REGION Network 138: GROUP 6 SAFE STOP 1 DEACTIVATE
   RUNG wire#powerrail
      Contact( "DB1018_SAFETY_TAGS".ALWAYS_ON )
      Coil( "DB1018_SAFETY_TAGS".GROUP_6_E20.SS1_Deactivate )
   END_RUNG
   // the same network as SCL:
   "DB1018_SAFETY_TAGS".GROUP_6_E20.SS1_Deactivate := "DB1018_SAFETY_TAGS".ALWAYS_ON;
END_REGION

REGION Network 139: DESELECT SAFE STOP 1
   RUNG wire#powerrail
      Contact( "DB1018_SAFETY_TAGS".GROUP_6_E20.SS1_Deactivate )
      Coil( "E20_SAFETY_OUT".Deselect_SS1 )
   END_RUNG
   // the same network as SCL:
   "E20_SAFETY_OUT".Deselect_SS1 := "DB1018_SAFETY_TAGS".GROUP_6_E20.SS1_Deactivate;
END_REGION

REGION Network 140: GROUP 6 SAFE STOP 2 DEACTIVATE
   RUNG wire#powerrail
      Contact( "DB1018_SAFETY_TAGS".E_STOP_OK )
      wire#w1
      Coil( "DB1018_SAFETY_TAGS".GROUP_6_E20.SS2_Deactivate )
   END_RUNG
   RUNG wire#powerrail
      Contact( "DB1018_SAFETY_TAGS".SAFE_DOORS_U02_CLOSED_AND_LOCKED )
   END_RUNG wire#w1
   // the same network as SCL:
   "DB1018_SAFETY_TAGS".GROUP_6_E20.SS2_Deactivate := "DB1018_SAFETY_TAGS".E_STOP_OK OR "DB1018_SAFETY_TAGS".SAFE_DOORS_U02_CLOSED_AND_LOCKED;
END_REGION

REGION Network 141: DESELECT SAFE STOP 2
   RUNG wire#powerrail
      Contact( "DB1018_SAFETY_TAGS".GROUP_6_E20.SS2_Deactivate )
      Coil( "E20_SAFETY_OUT".Deselect_SS2 )
   END_RUNG
   // the same network as SCL:
   "E20_SAFETY_OUT".Deselect_SS2 := "DB1018_SAFETY_TAGS".GROUP_6_E20.SS2_Deactivate;
END_REGION

REGION Network 142: GROUP 6 SAFE STOP 2 EXTENDED DEACTIVATE
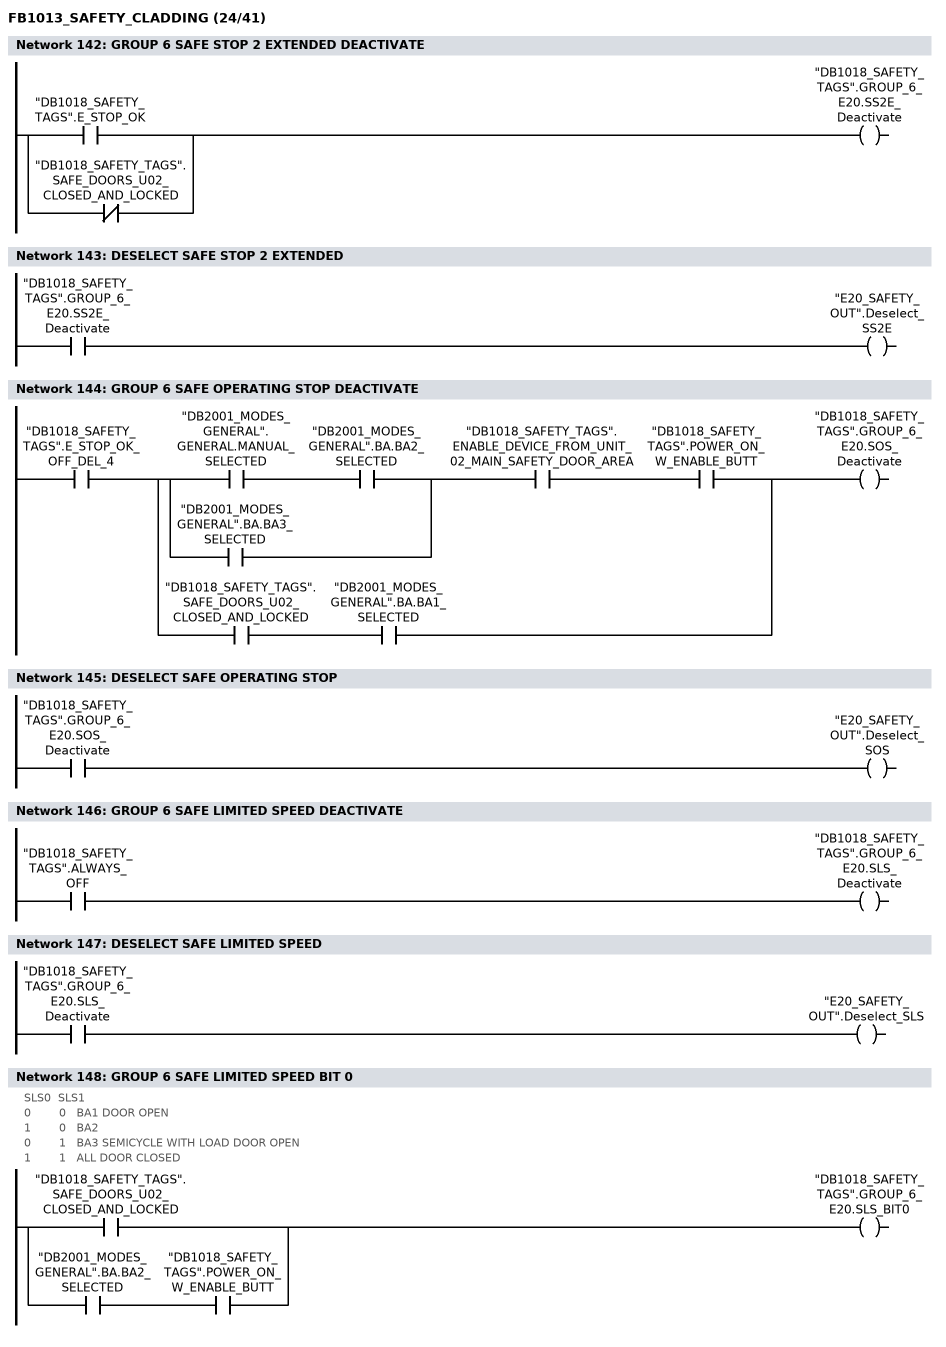
   RUNG wire#powerrail
      Contact( "DB1018_SAFETY_TAGS".E_STOP_OK )
      wire#w1
      Coil( "DB1018_SAFETY_TAGS".GROUP_6_E20.SS2E_Deactivate )
   END_RUNG
   RUNG wire#powerrail
      I_Contact( "DB1018_SAFETY_TAGS".SAFE_DOORS_U02_CLOSED_AND_LOCKED )
   END_RUNG wire#w1
   // the same network as SCL:
   "DB1018_SAFETY_TAGS".GROUP_6_E20.SS2E_Deactivate := "DB1018_SAFETY_TAGS".E_STOP_OK OR NOT "DB1018_SAFETY_TAGS".SAFE_DOORS_U02_CLOSED_AND_LOCKED;
END_REGION

REGION Network 143: DESELECT SAFE STOP 2 EXTENDED
   RUNG wire#powerrail
      Contact( "DB1018_SAFETY_TAGS".GROUP_6_E20.SS2E_Deactivate )
      Coil( "E20_SAFETY_OUT".Deselect_SS2E )
   END_RUNG
   // the same network as SCL:
   "E20_SAFETY_OUT".Deselect_SS2E := "DB1018_SAFETY_TAGS".GROUP_6_E20.SS2E_Deactivate;
END_REGION

REGION Network 144: GROUP 6 SAFE OPERATING STOP DEACTIVATE
   RUNG wire#powerrail
      Contact( "DB1018_SAFETY_TAGS".E_STOP_OK_OFF_DEL_4 )
      wire#w1
      Contact( "DB2001_MODES_GENERAL".GENERAL.MANUAL_SELECTED )
      Contact( "DB2001_MODES_GENERAL".BA.BA2_SELECTED )
      wire#w2
      Contact( "DB1018_SAFETY_TAGS".ENABLE_DEVICE_FROM_UNIT_02_MAIN_SAFETY_DOOR_AREA )
      Contact( "DB1018_SAFETY_TAGS".POWER_ON_W_ENABLE_BUTT )
      wire#w3
      Coil( "DB1018_SAFETY_TAGS".GROUP_6_E20.SOS_Deactivate )
   END_RUNG
   RUNG wire#w1
      Contact( "DB2001_MODES_GENERAL".BA.BA3_SELECTED )
   END_RUNG wire#w2
   RUNG wire#w1
      Contact( "DB1018_SAFETY_TAGS".SAFE_DOORS_U02_CLOSED_AND_LOCKED )
      Contact( "DB2001_MODES_GENERAL".BA.BA1_SELECTED )
   END_RUNG wire#w3
   // the same network as SCL:
   "DB1018_SAFETY_TAGS".GROUP_6_E20.SOS_Deactivate := "DB1018_SAFETY_TAGS".E_STOP_OK_OFF_DEL_4 AND (((("DB2001_MODES_GENERAL".GENERAL.MANUAL_SELECTED AND "DB2001_MODES_GENERAL".BA.BA2_SELECTED) OR "DB2001_MODES_GENERAL".BA.BA3_SELECTED) AND "DB1018_SAFETY_TAGS".ENABLE_DEVICE_FROM_UNIT_02_MAIN_SAFETY_DOOR_AREA AND "DB1018_SAFETY_TAGS".POWER_ON_W_ENABLE_BUTT) OR ("DB1018_SAFETY_TAGS".SAFE_DOORS_U02_CLOSED_AND_LOCKED AND "DB2001_MODES_GENERAL".BA.BA1_SELECTED));
END_REGION

REGION Network 145: DESELECT SAFE OPERATING STOP
   RUNG wire#powerrail
      Contact( "DB1018_SAFETY_TAGS".GROUP_6_E20.SOS_Deactivate )
      Coil( "E20_SAFETY_OUT".Deselect_SOS )
   END_RUNG
   // the same network as SCL:
   "E20_SAFETY_OUT".Deselect_SOS := "DB1018_SAFETY_TAGS".GROUP_6_E20.SOS_Deactivate;
END_REGION

REGION Network 146: GROUP 6 SAFE LIMITED SPEED DEACTIVATE
   RUNG wire#powerrail
      Contact( "DB1018_SAFETY_TAGS".ALWAYS_OFF )
      Coil( "DB1018_SAFETY_TAGS".GROUP_6_E20.SLS_Deactivate )
   END_RUNG
   // the same network as SCL:
   "DB1018_SAFETY_TAGS".GROUP_6_E20.SLS_Deactivate := "DB1018_SAFETY_TAGS".ALWAYS_OFF;
END_REGION

REGION Network 147: DESELECT SAFE LIMITED SPEED
   RUNG wire#powerrail
      Contact( "DB1018_SAFETY_TAGS".GROUP_6_E20.SLS_Deactivate )
      Coil( "E20_SAFETY_OUT".Deselect_SLS )
   END_RUNG
   // the same network as SCL:
   "E20_SAFETY_OUT".Deselect_SLS := "DB1018_SAFETY_TAGS".GROUP_6_E20.SLS_Deactivate;
END_REGION

REGION Network 148: GROUP 6 SAFE LIMITED SPEED BIT 0
   // SLS0  SLS1
   //    0        0   BA1 DOOR OPEN
   //    1        0   BA2
   //    0        1   BA3 SEMICYCLE WITH LOAD DOOR OPEN
   //    1        1   ALL DOOR CLOSED
   RUNG wire#powerrail
      Contact( "DB1018_SAFETY_TAGS".SAFE_DOORS_U02_CLOSED_AND_LOCKED )
      wire#w1
      Coil( "DB1018_SAFETY_TAGS".GROUP_6_E20.SLS_BIT0 )
   END_RUNG
   RUNG wire#powerrail
      Contact( "DB2001_MODES_GENERAL".BA.BA2_SELECTED )
      Contact( "DB1018_SAFETY_TAGS".POWER_ON_W_ENABLE_BUTT )
   END_RUNG wire#w1
   // the same network as SCL:
   "DB1018_SAFETY_TAGS".GROUP_6_E20.SLS_BIT0 := "DB1018_SAFETY_TAGS".SAFE_DOORS_U02_CLOSED_AND_LOCKED OR ("DB2001_MODES_GENERAL".BA.BA2_SELECTED AND "DB1018_SAFETY_TAGS".POWER_ON_W_ENABLE_BUTT);
END_REGION

REGION Network 149: SELECT SAFE LIMITED SPEED BIT 0
   // SLS0  SLS1
   //    0        0   BA1 DOOR OPEN
   //    1        0   BA2
   //    0        1   BA3 SEMICYCLE WITH LOAD DOOR OPEN
   //    1        1   ALL DOOR CLOSED
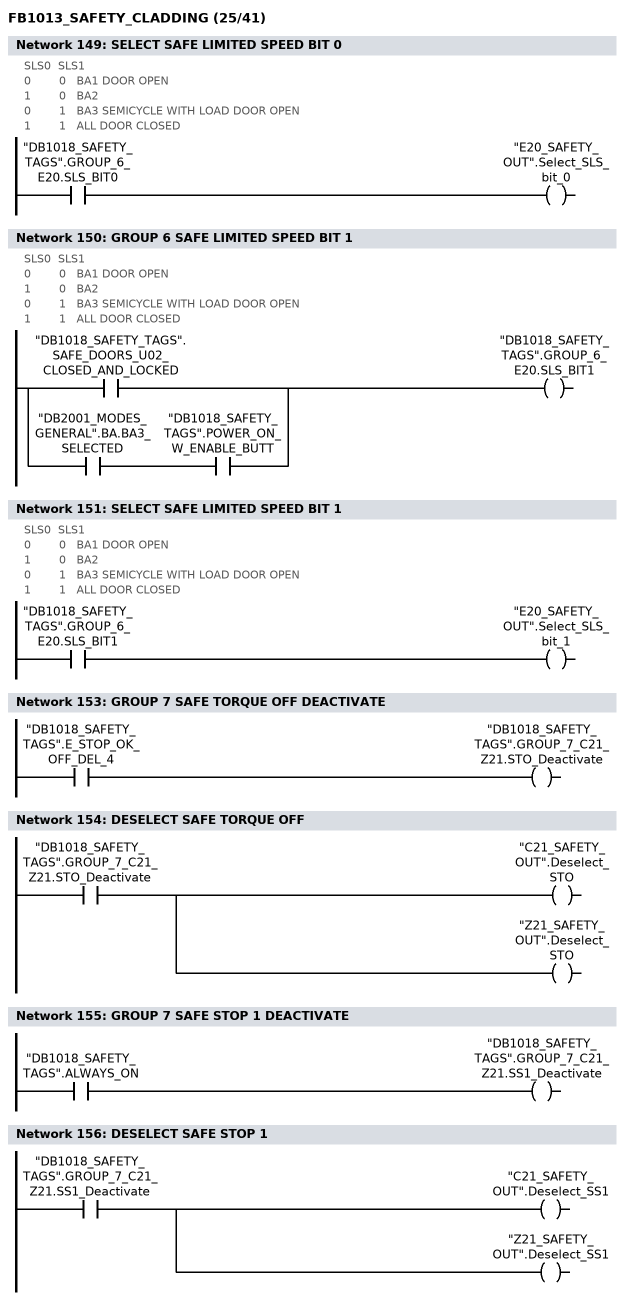
   RUNG wire#powerrail
      Contact( "DB1018_SAFETY_TAGS".GROUP_6_E20.SLS_BIT0 )
      Coil( "E20_SAFETY_OUT".Select_SLS_bit_0 )
   END_RUNG
   // the same network as SCL:
   "E20_SAFETY_OUT".Select_SLS_bit_0 := "DB1018_SAFETY_TAGS".GROUP_6_E20.SLS_BIT0;
END_REGION

REGION Network 150: GROUP 6 SAFE LIMITED SPEED BIT 1
   // SLS0  SLS1
   //    0        0   BA1 DOOR OPEN
   //    1        0   BA2
   //    0        1   BA3 SEMICYCLE WITH LOAD DOOR OPEN
   //    1        1   ALL DOOR CLOSED
   RUNG wire#powerrail
      Contact( "DB1018_SAFETY_TAGS".SAFE_DOORS_U02_CLOSED_AND_LOCKED )
      wire#w1
      Coil( "DB1018_SAFETY_TAGS".GROUP_6_E20.SLS_BIT1 )
   END_RUNG
   RUNG wire#powerrail
      Contact( "DB2001_MODES_GENERAL".BA.BA3_SELECTED )
      Contact( "DB1018_SAFETY_TAGS".POWER_ON_W_ENABLE_BUTT )
   END_RUNG wire#w1
   // the same network as SCL:
   "DB1018_SAFETY_TAGS".GROUP_6_E20.SLS_BIT1 := "DB1018_SAFETY_TAGS".SAFE_DOORS_U02_CLOSED_AND_LOCKED OR ("DB2001_MODES_GENERAL".BA.BA3_SELECTED AND "DB1018_SAFETY_TAGS".POWER_ON_W_ENABLE_BUTT);
END_REGION

REGION Network 151: SELECT SAFE LIMITED SPEED BIT 1
   // SLS0  SLS1
   //    0        0   BA1 DOOR OPEN
   //    1        0   BA2
   //    0        1   BA3 SEMICYCLE WITH LOAD DOOR OPEN
   //    1        1   ALL DOOR CLOSED
   RUNG wire#powerrail
      Contact( "DB1018_SAFETY_TAGS".GROUP_6_E20.SLS_BIT1 )
      Coil( "E20_SAFETY_OUT".Select_SLS_bit_1 )
   END_RUNG
   // the same network as SCL:
   "E20_SAFETY_OUT".Select_SLS_bit_1 := "DB1018_SAFETY_TAGS".GROUP_6_E20.SLS_BIT1;
END_REGION

REGION Network 152: *************** GROUP 7 - C21 / Z21 ***************
END_REGION

REGION Network 153: GROUP 7 SAFE TORQUE OFF DEACTIVATE
   RUNG wire#powerrail
      Contact( "DB1018_SAFETY_TAGS".E_STOP_OK_OFF_DEL_4 )
      Coil( "DB1018_SAFETY_TAGS".GROUP_7_C21_Z21.STO_Deactivate )
   END_RUNG
   // the same network as SCL:
   "DB1018_SAFETY_TAGS".GROUP_7_C21_Z21.STO_Deactivate := "DB1018_SAFETY_TAGS".E_STOP_OK_OFF_DEL_4;
END_REGION

REGION Network 154: DESELECT SAFE TORQUE OFF
   RUNG wire#powerrail
      Contact( "DB1018_SAFETY_TAGS".GROUP_7_C21_Z21.STO_Deactivate )
      wire#w1
      Coil( "C21_SAFETY_OUT".Deselect_STO )
   END_RUNG
   RUNG wire#w1
      Coil( "Z21_SAFETY_OUT".Deselect_STO )
   END_RUNG
   // the same network as SCL:
   "C21_SAFETY_OUT".Deselect_STO := "DB1018_SAFETY_TAGS".GROUP_7_C21_Z21.STO_Deactivate;
   "Z21_SAFETY_OUT".Deselect_STO := "DB1018_SAFETY_TAGS".GROUP_7_C21_Z21.STO_Deactivate;
END_REGION

REGION Network 155: GROUP 7 SAFE STOP 1 DEACTIVATE
   RUNG wire#powerrail
      Contact( "DB1018_SAFETY_TAGS".ALWAYS_ON )
      Coil( "DB1018_SAFETY_TAGS".GROUP_7_C21_Z21.SS1_Deactivate )
   END_RUNG
   // the same network as SCL:
   "DB1018_SAFETY_TAGS".GROUP_7_C21_Z21.SS1_Deactivate := "DB1018_SAFETY_TAGS".ALWAYS_ON;
END_REGION

REGION Network 156: DESELECT SAFE STOP 1
   RUNG wire#powerrail
      Contact( "DB1018_SAFETY_TAGS".GROUP_7_C21_Z21.SS1_Deactivate )
      wire#w1
      Coil( "C21_SAFETY_OUT".Deselect_SS1 )
   END_RUNG
   RUNG wire#w1
      Coil( "Z21_SAFETY_OUT".Deselect_SS1 )
   END_RUNG
   // the same network as SCL:
   "C21_SAFETY_OUT".Deselect_SS1 := "DB1018_SAFETY_TAGS".GROUP_7_C21_Z21.SS1_Deactivate;
   "Z21_SAFETY_OUT".Deselect_SS1 := "DB1018_SAFETY_TAGS".GROUP_7_C21_Z21.SS1_Deactivate;
END_REGION

REGION Network 157: GROUP 7 SAFE STOP 2 DEACTIVATE
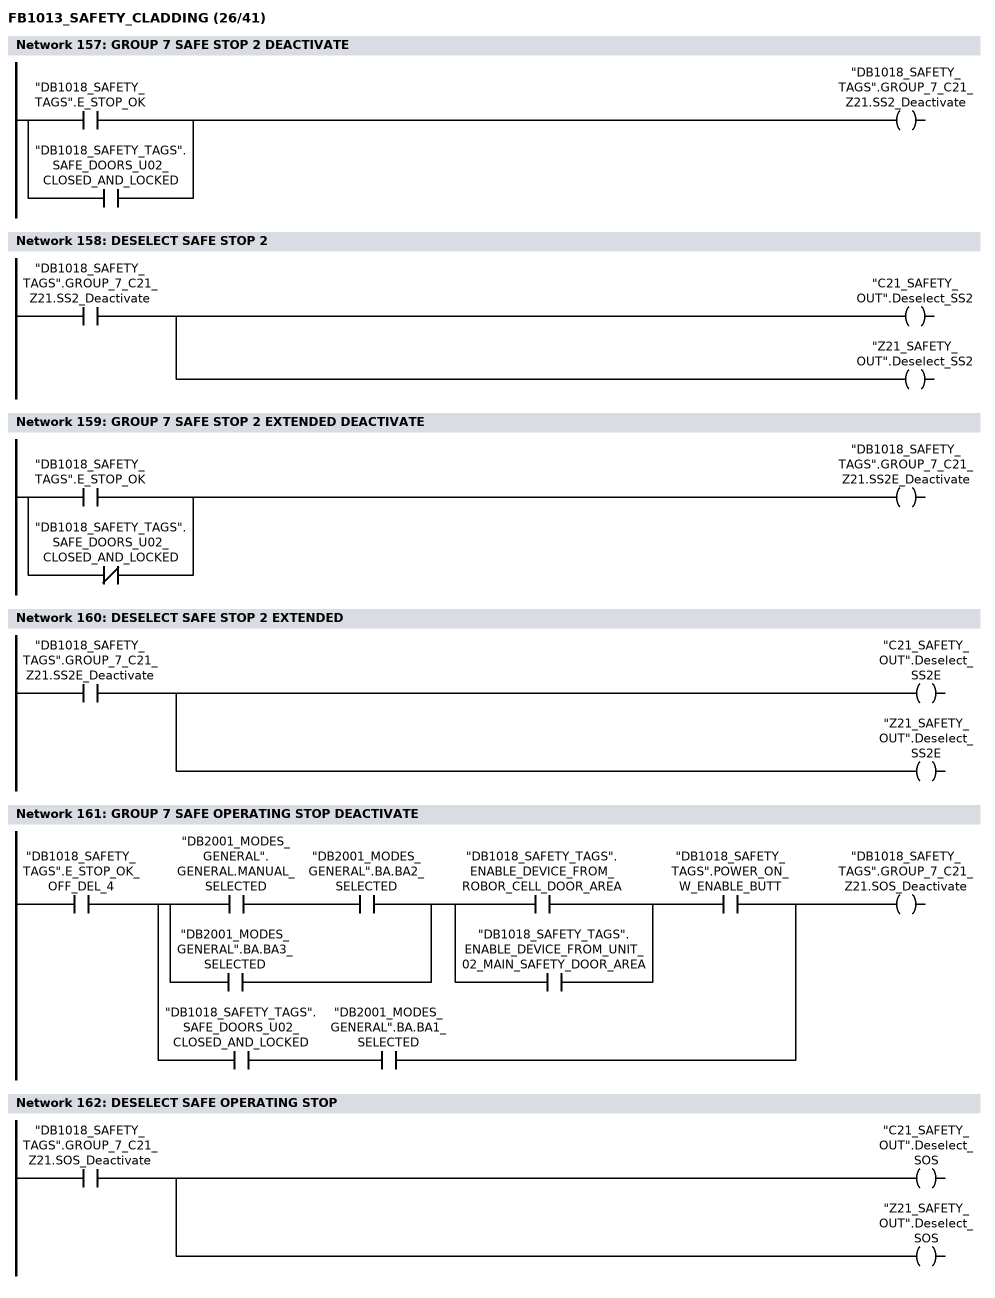
   RUNG wire#powerrail
      Contact( "DB1018_SAFETY_TAGS".E_STOP_OK )
      wire#w1
      Coil( "DB1018_SAFETY_TAGS".GROUP_7_C21_Z21.SS2_Deactivate )
   END_RUNG
   RUNG wire#powerrail
      Contact( "DB1018_SAFETY_TAGS".SAFE_DOORS_U02_CLOSED_AND_LOCKED )
   END_RUNG wire#w1
   // the same network as SCL:
   "DB1018_SAFETY_TAGS".GROUP_7_C21_Z21.SS2_Deactivate := "DB1018_SAFETY_TAGS".E_STOP_OK OR "DB1018_SAFETY_TAGS".SAFE_DOORS_U02_CLOSED_AND_LOCKED;
END_REGION

REGION Network 158: DESELECT SAFE STOP 2
   RUNG wire#powerrail
      Contact( "DB1018_SAFETY_TAGS".GROUP_7_C21_Z21.SS2_Deactivate )
      wire#w1
      Coil( "C21_SAFETY_OUT".Deselect_SS2 )
   END_RUNG
   RUNG wire#w1
      Coil( "Z21_SAFETY_OUT".Deselect_SS2 )
   END_RUNG
   // the same network as SCL:
   "C21_SAFETY_OUT".Deselect_SS2 := "DB1018_SAFETY_TAGS".GROUP_7_C21_Z21.SS2_Deactivate;
   "Z21_SAFETY_OUT".Deselect_SS2 := "DB1018_SAFETY_TAGS".GROUP_7_C21_Z21.SS2_Deactivate;
END_REGION

REGION Network 159: GROUP 7 SAFE STOP 2 EXTENDED DEACTIVATE
   RUNG wire#powerrail
      Contact( "DB1018_SAFETY_TAGS".E_STOP_OK )
      wire#w1
      Coil( "DB1018_SAFETY_TAGS".GROUP_7_C21_Z21.SS2E_Deactivate )
   END_RUNG
   RUNG wire#powerrail
      I_Contact( "DB1018_SAFETY_TAGS".SAFE_DOORS_U02_CLOSED_AND_LOCKED )
   END_RUNG wire#w1
   // the same network as SCL:
   "DB1018_SAFETY_TAGS".GROUP_7_C21_Z21.SS2E_Deactivate := "DB1018_SAFETY_TAGS".E_STOP_OK OR NOT "DB1018_SAFETY_TAGS".SAFE_DOORS_U02_CLOSED_AND_LOCKED;
END_REGION

REGION Network 160: DESELECT SAFE STOP 2 EXTENDED
   RUNG wire#powerrail
      Contact( "DB1018_SAFETY_TAGS".GROUP_7_C21_Z21.SS2E_Deactivate )
      wire#w1
      Coil( "C21_SAFETY_OUT".Deselect_SS2E )
   END_RUNG
   RUNG wire#w1
      Coil( "Z21_SAFETY_OUT".Deselect_SS2E )
   END_RUNG
   // the same network as SCL:
   "C21_SAFETY_OUT".Deselect_SS2E := "DB1018_SAFETY_TAGS".GROUP_7_C21_Z21.SS2E_Deactivate;
   "Z21_SAFETY_OUT".Deselect_SS2E := "DB1018_SAFETY_TAGS".GROUP_7_C21_Z21.SS2E_Deactivate;
END_REGION

REGION Network 161: GROUP 7 SAFE OPERATING STOP DEACTIVATE
   RUNG wire#powerrail
      Contact( "DB1018_SAFETY_TAGS".E_STOP_OK_OFF_DEL_4 )
      wire#w1
      Contact( "DB2001_MODES_GENERAL".GENERAL.MANUAL_SELECTED )
      Contact( "DB2001_MODES_GENERAL".BA.BA2_SELECTED )
      wire#w2
      Contact( "DB1018_SAFETY_TAGS".ENABLE_DEVICE_FROM_ROBOR_CELL_DOOR_AREA )
      wire#w3
      Contact( "DB1018_SAFETY_TAGS".POWER_ON_W_ENABLE_BUTT )
      wire#w4
      Coil( "DB1018_SAFETY_TAGS".GROUP_7_C21_Z21.SOS_Deactivate )
   END_RUNG
   RUNG wire#w1
      Contact( "DB2001_MODES_GENERAL".BA.BA3_SELECTED )
   END_RUNG wire#w2
   RUNG wire#w2
      Contact( "DB1018_SAFETY_TAGS".ENABLE_DEVICE_FROM_UNIT_02_MAIN_SAFETY_DOOR_AREA )
   END_RUNG wire#w3
   RUNG wire#w1
      Contact( "DB1018_SAFETY_TAGS".SAFE_DOORS_U02_CLOSED_AND_LOCKED )
      Contact( "DB2001_MODES_GENERAL".BA.BA1_SELECTED )
   END_RUNG wire#w4
   // the same network as SCL:
   "DB1018_SAFETY_TAGS".GROUP_7_C21_Z21.SOS_Deactivate := "DB1018_SAFETY_TAGS".E_STOP_OK_OFF_DEL_4 AND (((("DB2001_MODES_GENERAL".GENERAL.MANUAL_SELECTED AND "DB2001_MODES_GENERAL".BA.BA2_SELECTED) OR "DB2001_MODES_GENERAL".BA.BA3_SELECTED) AND ("DB1018_SAFETY_TAGS".ENABLE_DEVICE_FROM_ROBOR_CELL_DOOR_AREA OR "DB1018_SAFETY_TAGS".ENABLE_DEVICE_FROM_UNIT_02_MAIN_SAFETY_DOOR_AREA) AND "DB1018_SAFETY_TAGS".POWER_ON_W_ENABLE_BUTT) OR ("DB1018_SAFETY_TAGS".SAFE_DOORS_U02_CLOSED_AND_LOCKED AND "DB2001_MODES_GENERAL".BA.BA1_SELECTED));
END_REGION

REGION Network 162: DESELECT SAFE OPERATING STOP
   RUNG wire#powerrail
      Contact( "DB1018_SAFETY_TAGS".GROUP_7_C21_Z21.SOS_Deactivate )
      wire#w1
      Coil( "C21_SAFETY_OUT".Deselect_SOS )
   END_RUNG
   RUNG wire#w1
      Coil( "Z21_SAFETY_OUT".Deselect_SOS )
   END_RUNG
   // the same network as SCL:
   "C21_SAFETY_OUT".Deselect_SOS := "DB1018_SAFETY_TAGS".GROUP_7_C21_Z21.SOS_Deactivate;
   "Z21_SAFETY_OUT".Deselect_SOS := "DB1018_SAFETY_TAGS".GROUP_7_C21_Z21.SOS_Deactivate;
END_REGION

REGION Network 163: GROUP 7 SAFE LIMITED SPEED DEACTIVATE
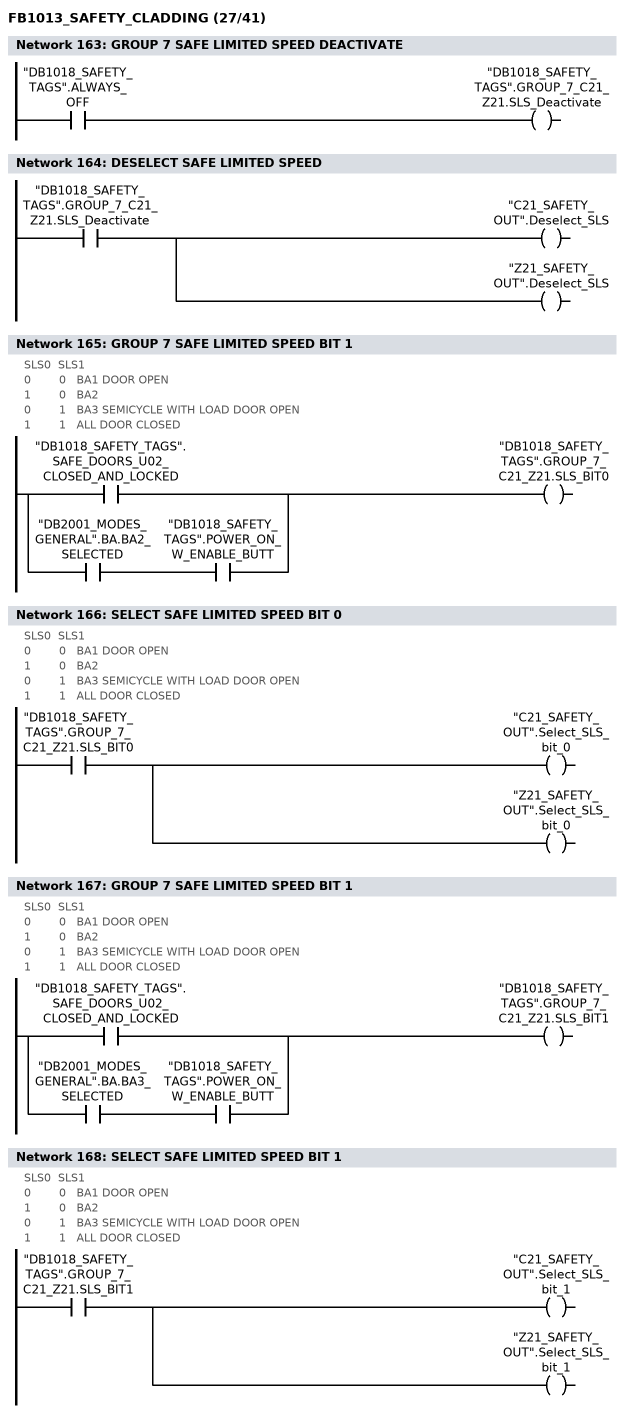
   RUNG wire#powerrail
      Contact( "DB1018_SAFETY_TAGS".ALWAYS_OFF )
      Coil( "DB1018_SAFETY_TAGS".GROUP_7_C21_Z21.SLS_Deactivate )
   END_RUNG
   // the same network as SCL:
   "DB1018_SAFETY_TAGS".GROUP_7_C21_Z21.SLS_Deactivate := "DB1018_SAFETY_TAGS".ALWAYS_OFF;
END_REGION

REGION Network 164: DESELECT SAFE LIMITED SPEED
   RUNG wire#powerrail
      Contact( "DB1018_SAFETY_TAGS".GROUP_7_C21_Z21.SLS_Deactivate )
      wire#w1
      Coil( "C21_SAFETY_OUT".Deselect_SLS )
   END_RUNG
   RUNG wire#w1
      Coil( "Z21_SAFETY_OUT".Deselect_SLS )
   END_RUNG
   // the same network as SCL:
   "C21_SAFETY_OUT".Deselect_SLS := "DB1018_SAFETY_TAGS".GROUP_7_C21_Z21.SLS_Deactivate;
   "Z21_SAFETY_OUT".Deselect_SLS := "DB1018_SAFETY_TAGS".GROUP_7_C21_Z21.SLS_Deactivate;
END_REGION

REGION Network 165: GROUP 7 SAFE LIMITED SPEED BIT 1
   // SLS0  SLS1
   //    0        0   BA1 DOOR OPEN
   //    1        0   BA2
   //    0        1   BA3 SEMICYCLE WITH LOAD DOOR OPEN
   //    1        1   ALL DOOR CLOSED
   RUNG wire#powerrail
      Contact( "DB1018_SAFETY_TAGS".SAFE_DOORS_U02_CLOSED_AND_LOCKED )
      wire#w1
      Coil( "DB1018_SAFETY_TAGS".GROUP_7_C21_Z21.SLS_BIT0 )
   END_RUNG
   RUNG wire#powerrail
      Contact( "DB2001_MODES_GENERAL".BA.BA2_SELECTED )
      Contact( "DB1018_SAFETY_TAGS".POWER_ON_W_ENABLE_BUTT )
   END_RUNG wire#w1
   // the same network as SCL:
   "DB1018_SAFETY_TAGS".GROUP_7_C21_Z21.SLS_BIT0 := "DB1018_SAFETY_TAGS".SAFE_DOORS_U02_CLOSED_AND_LOCKED OR ("DB2001_MODES_GENERAL".BA.BA2_SELECTED AND "DB1018_SAFETY_TAGS".POWER_ON_W_ENABLE_BUTT);
END_REGION

REGION Network 166: SELECT SAFE LIMITED SPEED BIT 0
   // SLS0  SLS1
   //    0        0   BA1 DOOR OPEN
   //    1        0   BA2
   //    0        1   BA3 SEMICYCLE WITH LOAD DOOR OPEN
   //    1        1   ALL DOOR CLOSED
   RUNG wire#powerrail
      Contact( "DB1018_SAFETY_TAGS".GROUP_7_C21_Z21.SLS_BIT0 )
      wire#w1
      Coil( "C21_SAFETY_OUT".Select_SLS_bit_0 )
   END_RUNG
   RUNG wire#w1
      Coil( "Z21_SAFETY_OUT".Select_SLS_bit_0 )
   END_RUNG
   // the same network as SCL:
   "C21_SAFETY_OUT".Select_SLS_bit_0 := "DB1018_SAFETY_TAGS".GROUP_7_C21_Z21.SLS_BIT0;
   "Z21_SAFETY_OUT".Select_SLS_bit_0 := "DB1018_SAFETY_TAGS".GROUP_7_C21_Z21.SLS_BIT0;
END_REGION

REGION Network 167: GROUP 7 SAFE LIMITED SPEED BIT 1
   // SLS0  SLS1
   //    0        0   BA1 DOOR OPEN
   //    1        0   BA2
   //    0        1   BA3 SEMICYCLE WITH LOAD DOOR OPEN
   //    1        1   ALL DOOR CLOSED
   RUNG wire#powerrail
      Contact( "DB1018_SAFETY_TAGS".SAFE_DOORS_U02_CLOSED_AND_LOCKED )
      wire#w1
      Coil( "DB1018_SAFETY_TAGS".GROUP_7_C21_Z21.SLS_BIT1 )
   END_RUNG
   RUNG wire#powerrail
      Contact( "DB2001_MODES_GENERAL".BA.BA3_SELECTED )
      Contact( "DB1018_SAFETY_TAGS".POWER_ON_W_ENABLE_BUTT )
   END_RUNG wire#w1
   // the same network as SCL:
   "DB1018_SAFETY_TAGS".GROUP_7_C21_Z21.SLS_BIT1 := "DB1018_SAFETY_TAGS".SAFE_DOORS_U02_CLOSED_AND_LOCKED OR ("DB2001_MODES_GENERAL".BA.BA3_SELECTED AND "DB1018_SAFETY_TAGS".POWER_ON_W_ENABLE_BUTT);
END_REGION

REGION Network 168: SELECT SAFE LIMITED SPEED BIT 1
   // SLS0  SLS1
   //    0        0   BA1 DOOR OPEN
   //    1        0   BA2
   //    0        1   BA3 SEMICYCLE WITH LOAD DOOR OPEN
   //    1        1   ALL DOOR CLOSED
   RUNG wire#powerrail
      Contact( "DB1018_SAFETY_TAGS".GROUP_7_C21_Z21.SLS_BIT1 )
      wire#w1
      Coil( "C21_SAFETY_OUT".Select_SLS_bit_1 )
   END_RUNG
   RUNG wire#w1
      Coil( "Z21_SAFETY_OUT".Select_SLS_bit_1 )
   END_RUNG
   // the same network as SCL:
   "C21_SAFETY_OUT".Select_SLS_bit_1 := "DB1018_SAFETY_TAGS".GROUP_7_C21_Z21.SLS_BIT1;
   "Z21_SAFETY_OUT".Select_SLS_bit_1 := "DB1018_SAFETY_TAGS".GROUP_7_C21_Z21.SLS_BIT1;
END_REGION

REGION Network 169: *************** GROUP 8 - C22 ***************
END_REGION

REGION Network 170: GROUP 8 SAFE TORQUE OFF DEACTIVATE
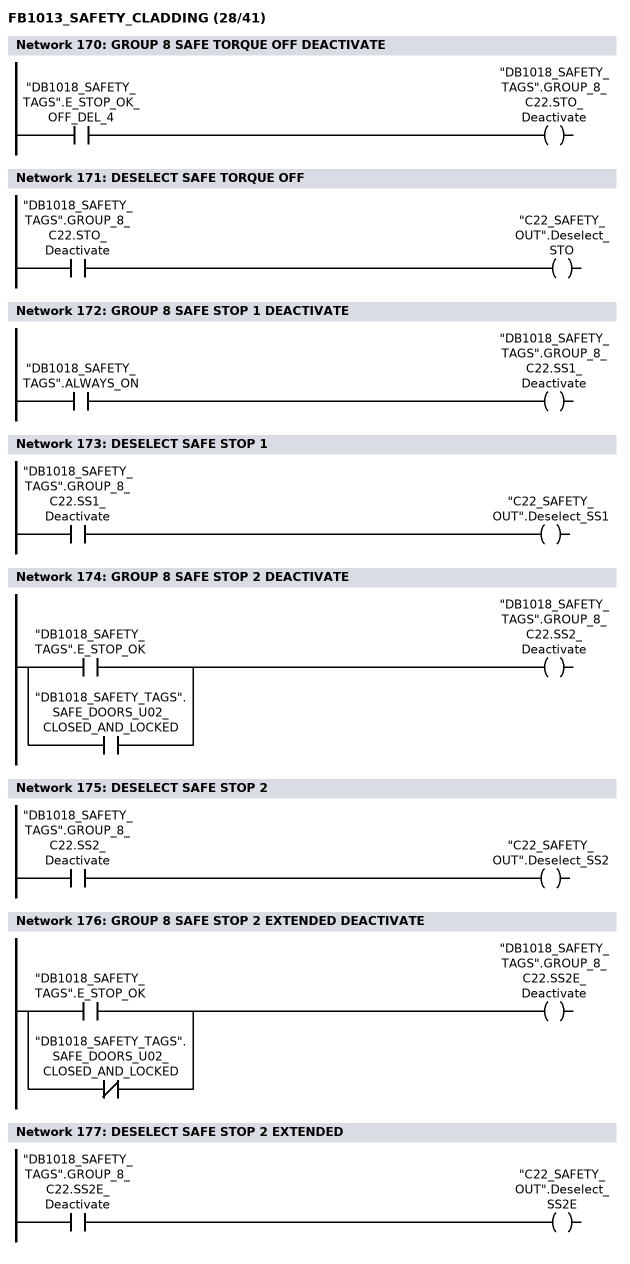
   RUNG wire#powerrail
      Contact( "DB1018_SAFETY_TAGS".E_STOP_OK_OFF_DEL_4 )
      Coil( "DB1018_SAFETY_TAGS".GROUP_8_C22.STO_Deactivate )
   END_RUNG
   // the same network as SCL:
   "DB1018_SAFETY_TAGS".GROUP_8_C22.STO_Deactivate := "DB1018_SAFETY_TAGS".E_STOP_OK_OFF_DEL_4;
END_REGION

REGION Network 171: DESELECT SAFE TORQUE OFF
   RUNG wire#powerrail
      Contact( "DB1018_SAFETY_TAGS".GROUP_8_C22.STO_Deactivate )
      Coil( "C22_SAFETY_OUT".Deselect_STO )
   END_RUNG
   // the same network as SCL:
   "C22_SAFETY_OUT".Deselect_STO := "DB1018_SAFETY_TAGS".GROUP_8_C22.STO_Deactivate;
END_REGION

REGION Network 172: GROUP 8 SAFE STOP 1 DEACTIVATE
   RUNG wire#powerrail
      Contact( "DB1018_SAFETY_TAGS".ALWAYS_ON )
      Coil( "DB1018_SAFETY_TAGS".GROUP_8_C22.SS1_Deactivate )
   END_RUNG
   // the same network as SCL:
   "DB1018_SAFETY_TAGS".GROUP_8_C22.SS1_Deactivate := "DB1018_SAFETY_TAGS".ALWAYS_ON;
END_REGION

REGION Network 173: DESELECT SAFE STOP 1
   RUNG wire#powerrail
      Contact( "DB1018_SAFETY_TAGS".GROUP_8_C22.SS1_Deactivate )
      Coil( "C22_SAFETY_OUT".Deselect_SS1 )
   END_RUNG
   // the same network as SCL:
   "C22_SAFETY_OUT".Deselect_SS1 := "DB1018_SAFETY_TAGS".GROUP_8_C22.SS1_Deactivate;
END_REGION

REGION Network 174: GROUP 8 SAFE STOP 2 DEACTIVATE
   RUNG wire#powerrail
      Contact( "DB1018_SAFETY_TAGS".E_STOP_OK )
      wire#w1
      Coil( "DB1018_SAFETY_TAGS".GROUP_8_C22.SS2_Deactivate )
   END_RUNG
   RUNG wire#powerrail
      Contact( "DB1018_SAFETY_TAGS".SAFE_DOORS_U02_CLOSED_AND_LOCKED )
   END_RUNG wire#w1
   // the same network as SCL:
   "DB1018_SAFETY_TAGS".GROUP_8_C22.SS2_Deactivate := "DB1018_SAFETY_TAGS".E_STOP_OK OR "DB1018_SAFETY_TAGS".SAFE_DOORS_U02_CLOSED_AND_LOCKED;
END_REGION

REGION Network 175: DESELECT SAFE STOP 2
   RUNG wire#powerrail
      Contact( "DB1018_SAFETY_TAGS".GROUP_8_C22.SS2_Deactivate )
      Coil( "C22_SAFETY_OUT".Deselect_SS2 )
   END_RUNG
   // the same network as SCL:
   "C22_SAFETY_OUT".Deselect_SS2 := "DB1018_SAFETY_TAGS".GROUP_8_C22.SS2_Deactivate;
END_REGION

REGION Network 176: GROUP 8 SAFE STOP 2 EXTENDED DEACTIVATE
   RUNG wire#powerrail
      Contact( "DB1018_SAFETY_TAGS".E_STOP_OK )
      wire#w1
      Coil( "DB1018_SAFETY_TAGS".GROUP_8_C22.SS2E_Deactivate )
   END_RUNG
   RUNG wire#powerrail
      I_Contact( "DB1018_SAFETY_TAGS".SAFE_DOORS_U02_CLOSED_AND_LOCKED )
   END_RUNG wire#w1
   // the same network as SCL:
   "DB1018_SAFETY_TAGS".GROUP_8_C22.SS2E_Deactivate := "DB1018_SAFETY_TAGS".E_STOP_OK OR NOT "DB1018_SAFETY_TAGS".SAFE_DOORS_U02_CLOSED_AND_LOCKED;
END_REGION

REGION Network 177: DESELECT SAFE STOP 2 EXTENDED
   RUNG wire#powerrail
      Contact( "DB1018_SAFETY_TAGS".GROUP_8_C22.SS2E_Deactivate )
      Coil( "C22_SAFETY_OUT".Deselect_SS2E )
   END_RUNG
   // the same network as SCL:
   "C22_SAFETY_OUT".Deselect_SS2E := "DB1018_SAFETY_TAGS".GROUP_8_C22.SS2E_Deactivate;
END_REGION

REGION Network 178: GROUP 8 SAFE OPERATING STOP DEACTIVATE
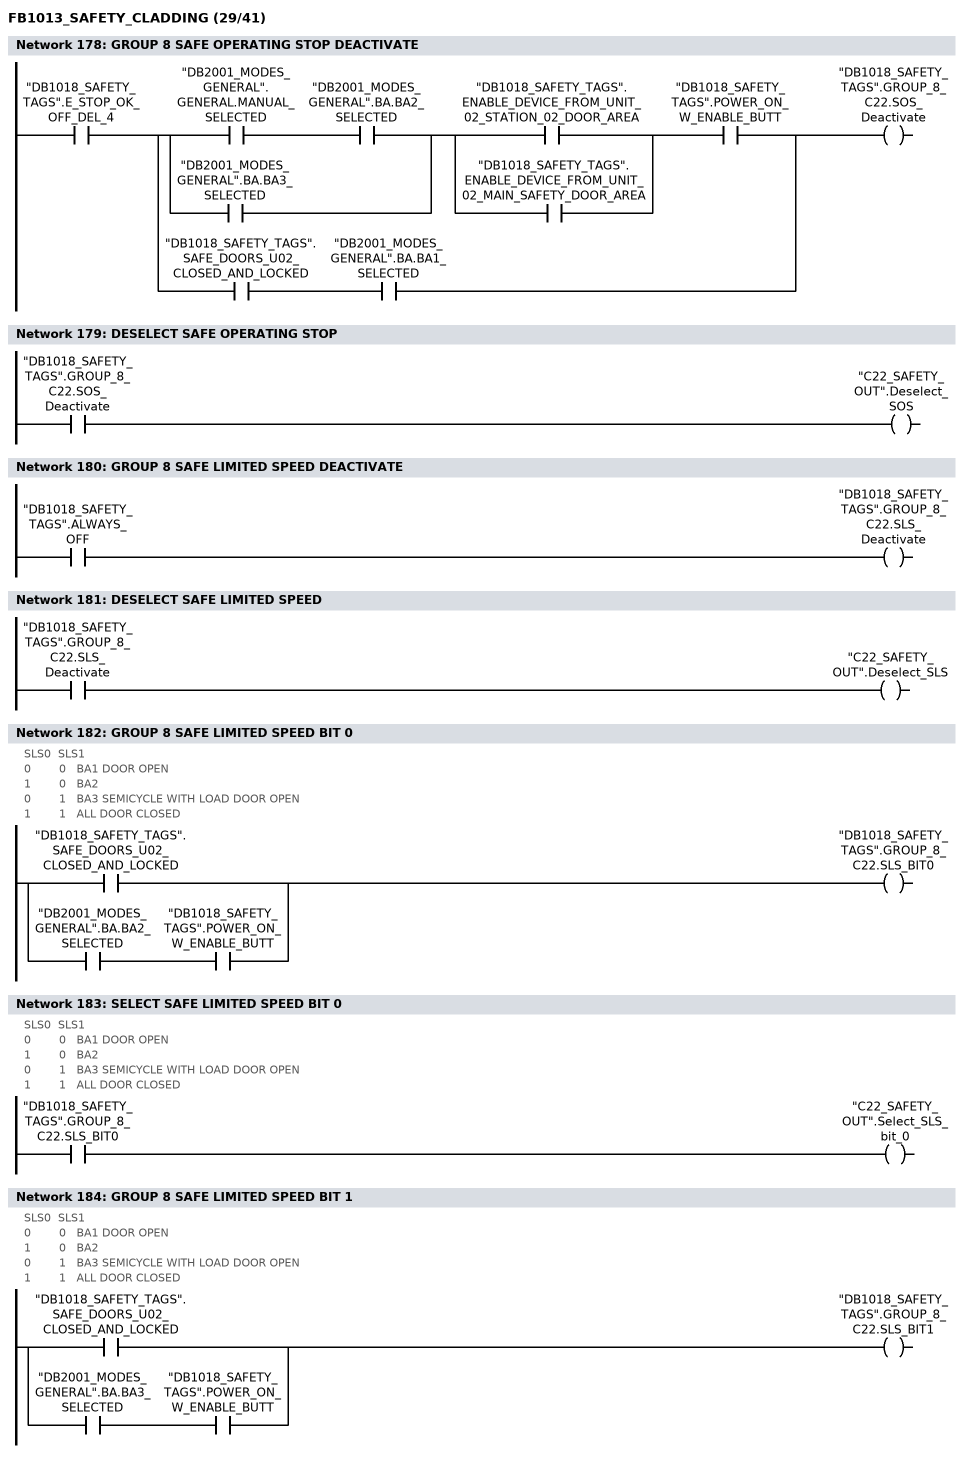
   RUNG wire#powerrail
      Contact( "DB1018_SAFETY_TAGS".E_STOP_OK_OFF_DEL_4 )
      wire#w1
      Contact( "DB2001_MODES_GENERAL".GENERAL.MANUAL_SELECTED )
      Contact( "DB2001_MODES_GENERAL".BA.BA2_SELECTED )
      wire#w2
      Contact( "DB1018_SAFETY_TAGS".ENABLE_DEVICE_FROM_UNIT_02_STATION_02_DOOR_AREA )
      wire#w3
      Contact( "DB1018_SAFETY_TAGS".POWER_ON_W_ENABLE_BUTT )
      wire#w4
      Coil( "DB1018_SAFETY_TAGS".GROUP_8_C22.SOS_Deactivate )
   END_RUNG
   RUNG wire#w1
      Contact( "DB2001_MODES_GENERAL".BA.BA3_SELECTED )
   END_RUNG wire#w2
   RUNG wire#w2
      Contact( "DB1018_SAFETY_TAGS".ENABLE_DEVICE_FROM_UNIT_02_MAIN_SAFETY_DOOR_AREA )
   END_RUNG wire#w3
   RUNG wire#w1
      Contact( "DB1018_SAFETY_TAGS".SAFE_DOORS_U02_CLOSED_AND_LOCKED )
      Contact( "DB2001_MODES_GENERAL".BA.BA1_SELECTED )
   END_RUNG wire#w4
   // the same network as SCL:
   "DB1018_SAFETY_TAGS".GROUP_8_C22.SOS_Deactivate := "DB1018_SAFETY_TAGS".E_STOP_OK_OFF_DEL_4 AND (((("DB2001_MODES_GENERAL".GENERAL.MANUAL_SELECTED AND "DB2001_MODES_GENERAL".BA.BA2_SELECTED) OR "DB2001_MODES_GENERAL".BA.BA3_SELECTED) AND ("DB1018_SAFETY_TAGS".ENABLE_DEVICE_FROM_UNIT_02_STATION_02_DOOR_AREA OR "DB1018_SAFETY_TAGS".ENABLE_DEVICE_FROM_UNIT_02_MAIN_SAFETY_DOOR_AREA) AND "DB1018_SAFETY_TAGS".POWER_ON_W_ENABLE_BUTT) OR ("DB1018_SAFETY_TAGS".SAFE_DOORS_U02_CLOSED_AND_LOCKED AND "DB2001_MODES_GENERAL".BA.BA1_SELECTED));
END_REGION

REGION Network 179: DESELECT SAFE OPERATING STOP
   RUNG wire#powerrail
      Contact( "DB1018_SAFETY_TAGS".GROUP_8_C22.SOS_Deactivate )
      Coil( "C22_SAFETY_OUT".Deselect_SOS )
   END_RUNG
   // the same network as SCL:
   "C22_SAFETY_OUT".Deselect_SOS := "DB1018_SAFETY_TAGS".GROUP_8_C22.SOS_Deactivate;
END_REGION

REGION Network 180: GROUP 8 SAFE LIMITED SPEED DEACTIVATE
   RUNG wire#powerrail
      Contact( "DB1018_SAFETY_TAGS".ALWAYS_OFF )
      Coil( "DB1018_SAFETY_TAGS".GROUP_8_C22.SLS_Deactivate )
   END_RUNG
   // the same network as SCL:
   "DB1018_SAFETY_TAGS".GROUP_8_C22.SLS_Deactivate := "DB1018_SAFETY_TAGS".ALWAYS_OFF;
END_REGION

REGION Network 181: DESELECT SAFE LIMITED SPEED
   RUNG wire#powerrail
      Contact( "DB1018_SAFETY_TAGS".GROUP_8_C22.SLS_Deactivate )
      Coil( "C22_SAFETY_OUT".Deselect_SLS )
   END_RUNG
   // the same network as SCL:
   "C22_SAFETY_OUT".Deselect_SLS := "DB1018_SAFETY_TAGS".GROUP_8_C22.SLS_Deactivate;
END_REGION

REGION Network 182: GROUP 8 SAFE LIMITED SPEED BIT 0
   // SLS0  SLS1
   //    0        0   BA1 DOOR OPEN
   //    1        0   BA2
   //    0        1   BA3 SEMICYCLE WITH LOAD DOOR OPEN
   //    1        1   ALL DOOR CLOSED
   RUNG wire#powerrail
      Contact( "DB1018_SAFETY_TAGS".SAFE_DOORS_U02_CLOSED_AND_LOCKED )
      wire#w1
      Coil( "DB1018_SAFETY_TAGS".GROUP_8_C22.SLS_BIT0 )
   END_RUNG
   RUNG wire#powerrail
      Contact( "DB2001_MODES_GENERAL".BA.BA2_SELECTED )
      Contact( "DB1018_SAFETY_TAGS".POWER_ON_W_ENABLE_BUTT )
   END_RUNG wire#w1
   // the same network as SCL:
   "DB1018_SAFETY_TAGS".GROUP_8_C22.SLS_BIT0 := "DB1018_SAFETY_TAGS".SAFE_DOORS_U02_CLOSED_AND_LOCKED OR ("DB2001_MODES_GENERAL".BA.BA2_SELECTED AND "DB1018_SAFETY_TAGS".POWER_ON_W_ENABLE_BUTT);
END_REGION

REGION Network 183: SELECT SAFE LIMITED SPEED BIT 0
   // SLS0  SLS1
   //    0        0   BA1 DOOR OPEN
   //    1        0   BA2
   //    0        1   BA3 SEMICYCLE WITH LOAD DOOR OPEN
   //    1        1   ALL DOOR CLOSED
   RUNG wire#powerrail
      Contact( "DB1018_SAFETY_TAGS".GROUP_8_C22.SLS_BIT0 )
      Coil( "C22_SAFETY_OUT".Select_SLS_bit_0 )
   END_RUNG
   // the same network as SCL:
   "C22_SAFETY_OUT".Select_SLS_bit_0 := "DB1018_SAFETY_TAGS".GROUP_8_C22.SLS_BIT0;
END_REGION

REGION Network 184: GROUP 8 SAFE LIMITED SPEED BIT 1
   // SLS0  SLS1
   //    0        0   BA1 DOOR OPEN
   //    1        0   BA2
   //    0        1   BA3 SEMICYCLE WITH LOAD DOOR OPEN
   //    1        1   ALL DOOR CLOSED
   RUNG wire#powerrail
      Contact( "DB1018_SAFETY_TAGS".SAFE_DOORS_U02_CLOSED_AND_LOCKED )
      wire#w1
      Coil( "DB1018_SAFETY_TAGS".GROUP_8_C22.SLS_BIT1 )
   END_RUNG
   RUNG wire#powerrail
      Contact( "DB2001_MODES_GENERAL".BA.BA3_SELECTED )
      Contact( "DB1018_SAFETY_TAGS".POWER_ON_W_ENABLE_BUTT )
   END_RUNG wire#w1
   // the same network as SCL:
   "DB1018_SAFETY_TAGS".GROUP_8_C22.SLS_BIT1 := "DB1018_SAFETY_TAGS".SAFE_DOORS_U02_CLOSED_AND_LOCKED OR ("DB2001_MODES_GENERAL".BA.BA3_SELECTED AND "DB1018_SAFETY_TAGS".POWER_ON_W_ENABLE_BUTT);
END_REGION

REGION Network 185: SELECT SAFE LIMITED SPEED BIT 1
   // SLS0  SLS1
   //    0        0   BA1 DOOR OPEN
   //    1        0   BA2
   //    0        1   BA3 SEMICYCLE WITH LOAD DOOR OPEN
   //    1        1   ALL DOOR CLOSED
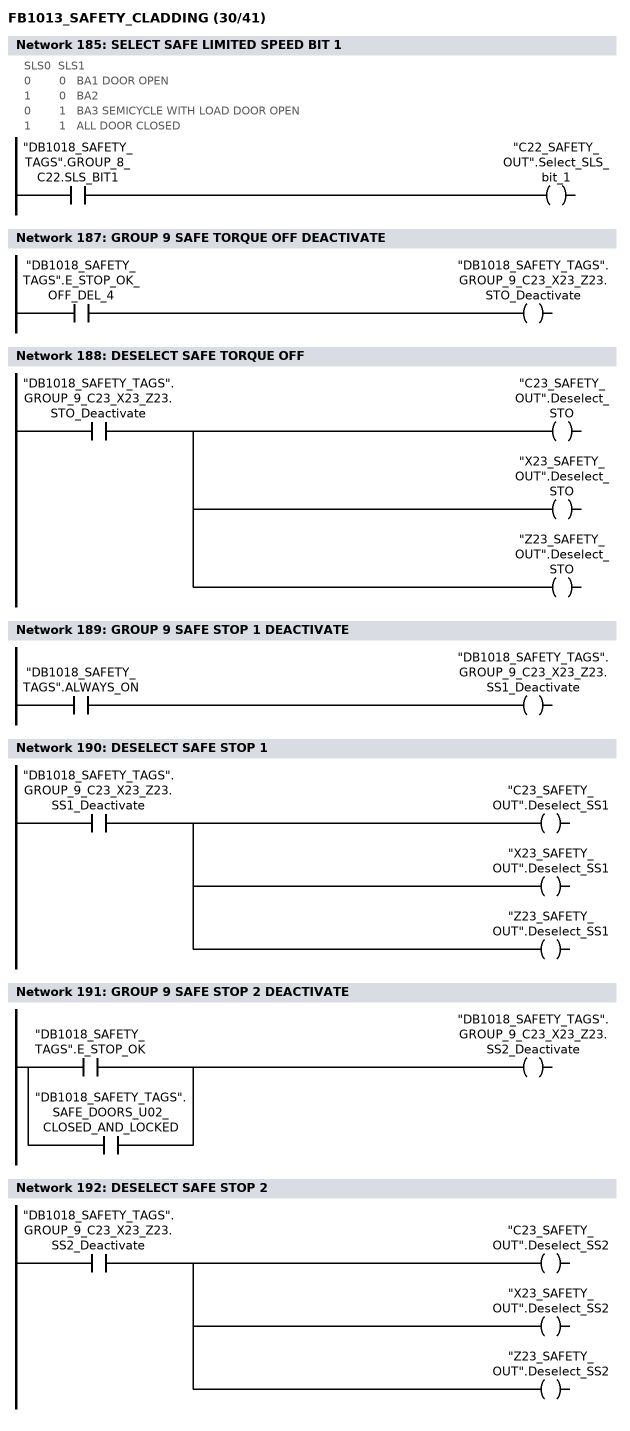
   RUNG wire#powerrail
      Contact( "DB1018_SAFETY_TAGS".GROUP_8_C22.SLS_BIT1 )
      Coil( "C22_SAFETY_OUT".Select_SLS_bit_1 )
   END_RUNG
   // the same network as SCL:
   "C22_SAFETY_OUT".Select_SLS_bit_1 := "DB1018_SAFETY_TAGS".GROUP_8_C22.SLS_BIT1;
END_REGION

REGION Network 186: *************** GROUP 9 - C23 / X23 / Z23 ***************
END_REGION

REGION Network 187: GROUP 9 SAFE TORQUE OFF DEACTIVATE
   RUNG wire#powerrail
      Contact( "DB1018_SAFETY_TAGS".E_STOP_OK_OFF_DEL_4 )
      Coil( "DB1018_SAFETY_TAGS".GROUP_9_C23_X23_Z23.STO_Deactivate )
   END_RUNG
   // the same network as SCL:
   "DB1018_SAFETY_TAGS".GROUP_9_C23_X23_Z23.STO_Deactivate := "DB1018_SAFETY_TAGS".E_STOP_OK_OFF_DEL_4;
END_REGION

REGION Network 188: DESELECT SAFE TORQUE OFF
   RUNG wire#powerrail
      Contact( "DB1018_SAFETY_TAGS".GROUP_9_C23_X23_Z23.STO_Deactivate )
      wire#w1
      Coil( "C23_SAFETY_OUT".Deselect_STO )
   END_RUNG
   RUNG wire#w1
      Coil( "X23_SAFETY_OUT".Deselect_STO )
   END_RUNG
   RUNG wire#w1
      Coil( "Z23_SAFETY_OUT".Deselect_STO )
   END_RUNG
   // the same network as SCL:
   "C23_SAFETY_OUT".Deselect_STO := "DB1018_SAFETY_TAGS".GROUP_9_C23_X23_Z23.STO_Deactivate;
   "X23_SAFETY_OUT".Deselect_STO := "DB1018_SAFETY_TAGS".GROUP_9_C23_X23_Z23.STO_Deactivate;
   "Z23_SAFETY_OUT".Deselect_STO := "DB1018_SAFETY_TAGS".GROUP_9_C23_X23_Z23.STO_Deactivate;
END_REGION

REGION Network 189: GROUP 9 SAFE STOP 1 DEACTIVATE
   RUNG wire#powerrail
      Contact( "DB1018_SAFETY_TAGS".ALWAYS_ON )
      Coil( "DB1018_SAFETY_TAGS".GROUP_9_C23_X23_Z23.SS1_Deactivate )
   END_RUNG
   // the same network as SCL:
   "DB1018_SAFETY_TAGS".GROUP_9_C23_X23_Z23.SS1_Deactivate := "DB1018_SAFETY_TAGS".ALWAYS_ON;
END_REGION

REGION Network 190: DESELECT SAFE STOP 1
   RUNG wire#powerrail
      Contact( "DB1018_SAFETY_TAGS".GROUP_9_C23_X23_Z23.SS1_Deactivate )
      wire#w1
      Coil( "C23_SAFETY_OUT".Deselect_SS1 )
   END_RUNG
   RUNG wire#w1
      Coil( "X23_SAFETY_OUT".Deselect_SS1 )
   END_RUNG
   RUNG wire#w1
      Coil( "Z23_SAFETY_OUT".Deselect_SS1 )
   END_RUNG
   // the same network as SCL:
   "C23_SAFETY_OUT".Deselect_SS1 := "DB1018_SAFETY_TAGS".GROUP_9_C23_X23_Z23.SS1_Deactivate;
   "X23_SAFETY_OUT".Deselect_SS1 := "DB1018_SAFETY_TAGS".GROUP_9_C23_X23_Z23.SS1_Deactivate;
   "Z23_SAFETY_OUT".Deselect_SS1 := "DB1018_SAFETY_TAGS".GROUP_9_C23_X23_Z23.SS1_Deactivate;
END_REGION

REGION Network 191: GROUP 9 SAFE STOP 2 DEACTIVATE
   RUNG wire#powerrail
      Contact( "DB1018_SAFETY_TAGS".E_STOP_OK )
      wire#w1
      Coil( "DB1018_SAFETY_TAGS".GROUP_9_C23_X23_Z23.SS2_Deactivate )
   END_RUNG
   RUNG wire#powerrail
      Contact( "DB1018_SAFETY_TAGS".SAFE_DOORS_U02_CLOSED_AND_LOCKED )
   END_RUNG wire#w1
   // the same network as SCL:
   "DB1018_SAFETY_TAGS".GROUP_9_C23_X23_Z23.SS2_Deactivate := "DB1018_SAFETY_TAGS".E_STOP_OK OR "DB1018_SAFETY_TAGS".SAFE_DOORS_U02_CLOSED_AND_LOCKED;
END_REGION

REGION Network 192: DESELECT SAFE STOP 2
   RUNG wire#powerrail
      Contact( "DB1018_SAFETY_TAGS".GROUP_9_C23_X23_Z23.SS2_Deactivate )
      wire#w1
      Coil( "C23_SAFETY_OUT".Deselect_SS2 )
   END_RUNG
   RUNG wire#w1
      Coil( "X23_SAFETY_OUT".Deselect_SS2 )
   END_RUNG
   RUNG wire#w1
      Coil( "Z23_SAFETY_OUT".Deselect_SS2 )
   END_RUNG
   // the same network as SCL:
   "C23_SAFETY_OUT".Deselect_SS2 := "DB1018_SAFETY_TAGS".GROUP_9_C23_X23_Z23.SS2_Deactivate;
   "X23_SAFETY_OUT".Deselect_SS2 := "DB1018_SAFETY_TAGS".GROUP_9_C23_X23_Z23.SS2_Deactivate;
   "Z23_SAFETY_OUT".Deselect_SS2 := "DB1018_SAFETY_TAGS".GROUP_9_C23_X23_Z23.SS2_Deactivate;
END_REGION

REGION Network 193: GROUP 9 SAFE STOP 2 EXTENDED DEACTIVATE
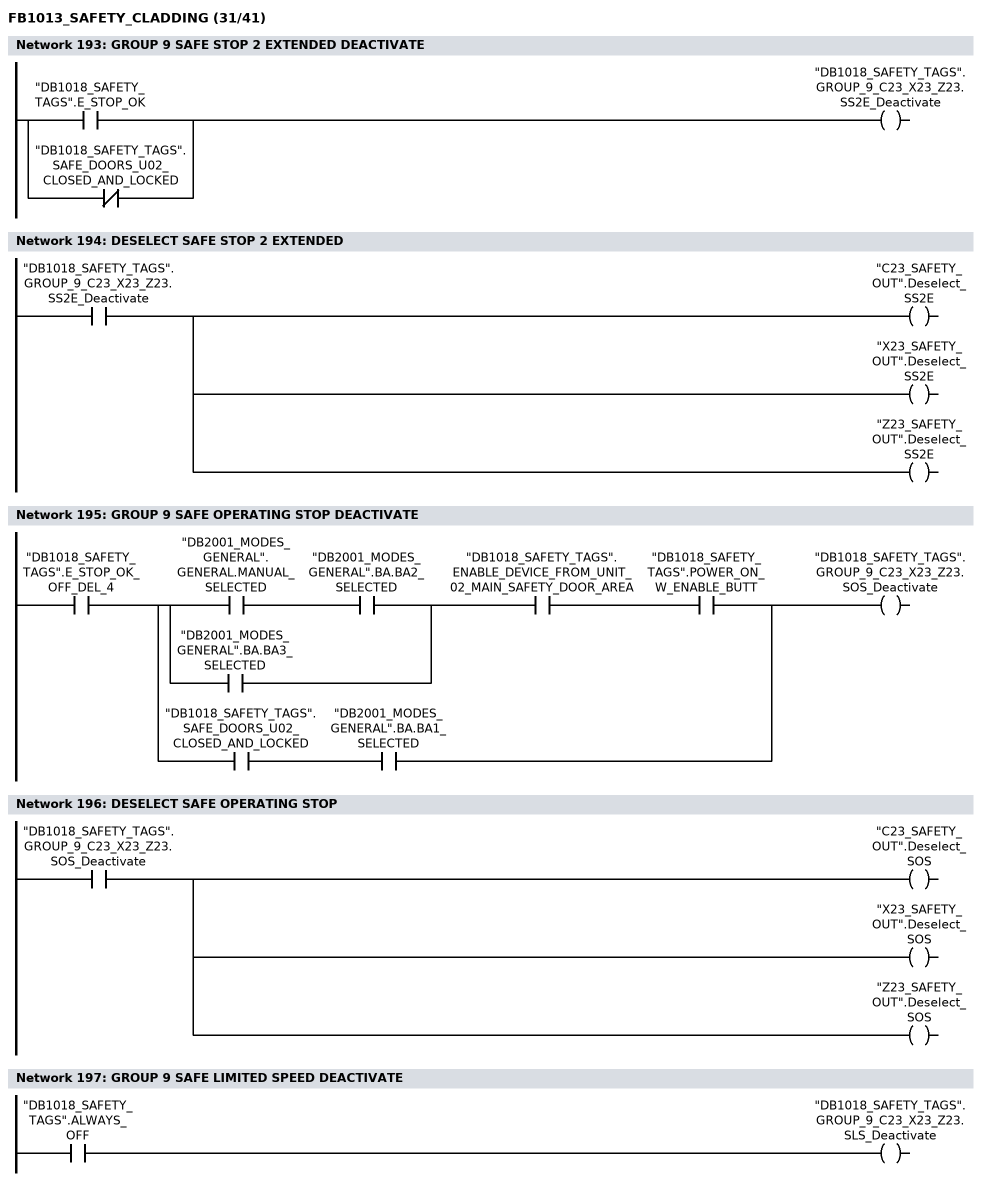
   RUNG wire#powerrail
      Contact( "DB1018_SAFETY_TAGS".E_STOP_OK )
      wire#w1
      Coil( "DB1018_SAFETY_TAGS".GROUP_9_C23_X23_Z23.SS2E_Deactivate )
   END_RUNG
   RUNG wire#powerrail
      I_Contact( "DB1018_SAFETY_TAGS".SAFE_DOORS_U02_CLOSED_AND_LOCKED )
   END_RUNG wire#w1
   // the same network as SCL:
   "DB1018_SAFETY_TAGS".GROUP_9_C23_X23_Z23.SS2E_Deactivate := "DB1018_SAFETY_TAGS".E_STOP_OK OR NOT "DB1018_SAFETY_TAGS".SAFE_DOORS_U02_CLOSED_AND_LOCKED;
END_REGION

REGION Network 194: DESELECT SAFE STOP 2 EXTENDED
   RUNG wire#powerrail
      Contact( "DB1018_SAFETY_TAGS".GROUP_9_C23_X23_Z23.SS2E_Deactivate )
      wire#w1
      Coil( "C23_SAFETY_OUT".Deselect_SS2E )
   END_RUNG
   RUNG wire#w1
      Coil( "X23_SAFETY_OUT".Deselect_SS2E )
   END_RUNG
   RUNG wire#w1
      Coil( "Z23_SAFETY_OUT".Deselect_SS2E )
   END_RUNG
   // the same network as SCL:
   "C23_SAFETY_OUT".Deselect_SS2E := "DB1018_SAFETY_TAGS".GROUP_9_C23_X23_Z23.SS2E_Deactivate;
   "X23_SAFETY_OUT".Deselect_SS2E := "DB1018_SAFETY_TAGS".GROUP_9_C23_X23_Z23.SS2E_Deactivate;
   "Z23_SAFETY_OUT".Deselect_SS2E := "DB1018_SAFETY_TAGS".GROUP_9_C23_X23_Z23.SS2E_Deactivate;
END_REGION

REGION Network 195: GROUP 9 SAFE OPERATING STOP DEACTIVATE
   RUNG wire#powerrail
      Contact( "DB1018_SAFETY_TAGS".E_STOP_OK_OFF_DEL_4 )
      wire#w1
      Contact( "DB2001_MODES_GENERAL".GENERAL.MANUAL_SELECTED )
      Contact( "DB2001_MODES_GENERAL".BA.BA2_SELECTED )
      wire#w2
      Contact( "DB1018_SAFETY_TAGS".ENABLE_DEVICE_FROM_UNIT_02_MAIN_SAFETY_DOOR_AREA )
      Contact( "DB1018_SAFETY_TAGS".POWER_ON_W_ENABLE_BUTT )
      wire#w3
      Coil( "DB1018_SAFETY_TAGS".GROUP_9_C23_X23_Z23.SOS_Deactivate )
   END_RUNG
   RUNG wire#w1
      Contact( "DB2001_MODES_GENERAL".BA.BA3_SELECTED )
   END_RUNG wire#w2
   RUNG wire#w1
      Contact( "DB1018_SAFETY_TAGS".SAFE_DOORS_U02_CLOSED_AND_LOCKED )
      Contact( "DB2001_MODES_GENERAL".BA.BA1_SELECTED )
   END_RUNG wire#w3
   // the same network as SCL:
   "DB1018_SAFETY_TAGS".GROUP_9_C23_X23_Z23.SOS_Deactivate := "DB1018_SAFETY_TAGS".E_STOP_OK_OFF_DEL_4 AND (((("DB2001_MODES_GENERAL".GENERAL.MANUAL_SELECTED AND "DB2001_MODES_GENERAL".BA.BA2_SELECTED) OR "DB2001_MODES_GENERAL".BA.BA3_SELECTED) AND "DB1018_SAFETY_TAGS".ENABLE_DEVICE_FROM_UNIT_02_MAIN_SAFETY_DOOR_AREA AND "DB1018_SAFETY_TAGS".POWER_ON_W_ENABLE_BUTT) OR ("DB1018_SAFETY_TAGS".SAFE_DOORS_U02_CLOSED_AND_LOCKED AND "DB2001_MODES_GENERAL".BA.BA1_SELECTED));
END_REGION

REGION Network 196: DESELECT SAFE OPERATING STOP
   RUNG wire#powerrail
      Contact( "DB1018_SAFETY_TAGS".GROUP_9_C23_X23_Z23.SOS_Deactivate )
      wire#w1
      Coil( "C23_SAFETY_OUT".Deselect_SOS )
   END_RUNG
   RUNG wire#w1
      Coil( "X23_SAFETY_OUT".Deselect_SOS )
   END_RUNG
   RUNG wire#w1
      Coil( "Z23_SAFETY_OUT".Deselect_SOS )
   END_RUNG
   // the same network as SCL:
   "C23_SAFETY_OUT".Deselect_SOS := "DB1018_SAFETY_TAGS".GROUP_9_C23_X23_Z23.SOS_Deactivate;
   "X23_SAFETY_OUT".Deselect_SOS := "DB1018_SAFETY_TAGS".GROUP_9_C23_X23_Z23.SOS_Deactivate;
   "Z23_SAFETY_OUT".Deselect_SOS := "DB1018_SAFETY_TAGS".GROUP_9_C23_X23_Z23.SOS_Deactivate;
END_REGION

REGION Network 197: GROUP 9 SAFE LIMITED SPEED DEACTIVATE
   RUNG wire#powerrail
      Contact( "DB1018_SAFETY_TAGS".ALWAYS_OFF )
      Coil( "DB1018_SAFETY_TAGS".GROUP_9_C23_X23_Z23.SLS_Deactivate )
   END_RUNG
   // the same network as SCL:
   "DB1018_SAFETY_TAGS".GROUP_9_C23_X23_Z23.SLS_Deactivate := "DB1018_SAFETY_TAGS".ALWAYS_OFF;
END_REGION

REGION Network 198: DESELECT SAFE LIMITED SPEED
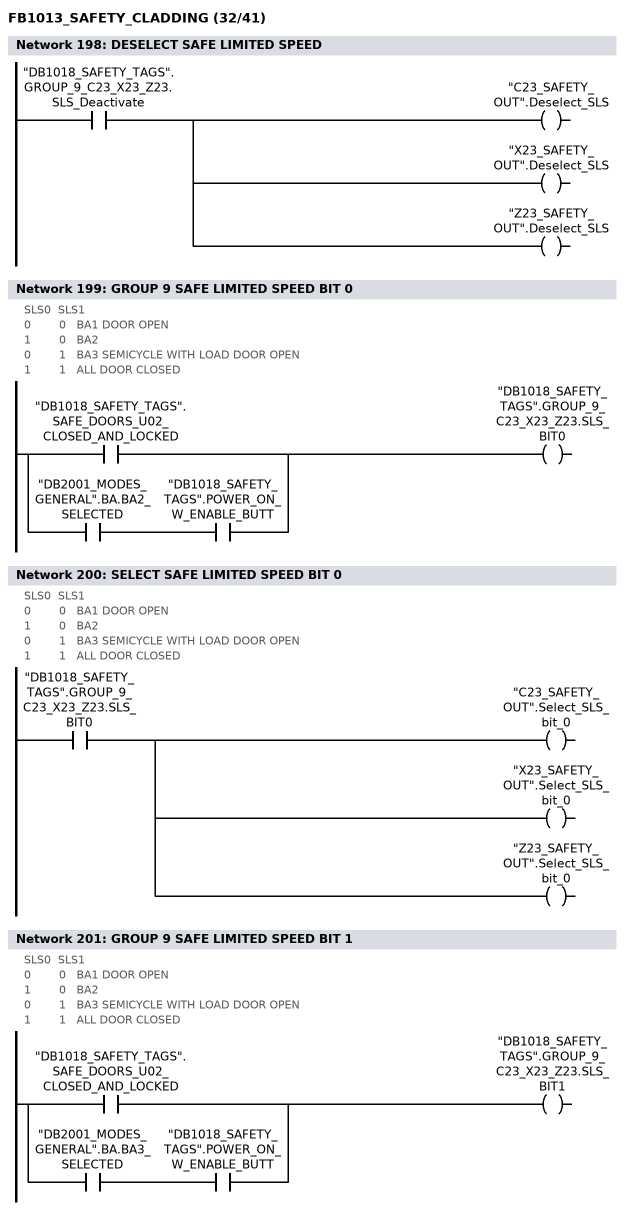
   RUNG wire#powerrail
      Contact( "DB1018_SAFETY_TAGS".GROUP_9_C23_X23_Z23.SLS_Deactivate )
      wire#w1
      Coil( "C23_SAFETY_OUT".Deselect_SLS )
   END_RUNG
   RUNG wire#w1
      Coil( "X23_SAFETY_OUT".Deselect_SLS )
   END_RUNG
   RUNG wire#w1
      Coil( "Z23_SAFETY_OUT".Deselect_SLS )
   END_RUNG
   // the same network as SCL:
   "C23_SAFETY_OUT".Deselect_SLS := "DB1018_SAFETY_TAGS".GROUP_9_C23_X23_Z23.SLS_Deactivate;
   "X23_SAFETY_OUT".Deselect_SLS := "DB1018_SAFETY_TAGS".GROUP_9_C23_X23_Z23.SLS_Deactivate;
   "Z23_SAFETY_OUT".Deselect_SLS := "DB1018_SAFETY_TAGS".GROUP_9_C23_X23_Z23.SLS_Deactivate;
END_REGION

REGION Network 199: GROUP 9 SAFE LIMITED SPEED BIT 0
   // SLS0  SLS1
   //    0        0   BA1 DOOR OPEN
   //    1        0   BA2
   //    0        1   BA3 SEMICYCLE WITH LOAD DOOR OPEN
   //    1        1   ALL DOOR CLOSED
   RUNG wire#powerrail
      Contact( "DB1018_SAFETY_TAGS".SAFE_DOORS_U02_CLOSED_AND_LOCKED )
      wire#w1
      Coil( "DB1018_SAFETY_TAGS".GROUP_9_C23_X23_Z23.SLS_BIT0 )
   END_RUNG
   RUNG wire#powerrail
      Contact( "DB2001_MODES_GENERAL".BA.BA2_SELECTED )
      Contact( "DB1018_SAFETY_TAGS".POWER_ON_W_ENABLE_BUTT )
   END_RUNG wire#w1
   // the same network as SCL:
   "DB1018_SAFETY_TAGS".GROUP_9_C23_X23_Z23.SLS_BIT0 := "DB1018_SAFETY_TAGS".SAFE_DOORS_U02_CLOSED_AND_LOCKED OR ("DB2001_MODES_GENERAL".BA.BA2_SELECTED AND "DB1018_SAFETY_TAGS".POWER_ON_W_ENABLE_BUTT);
END_REGION

REGION Network 200: SELECT SAFE LIMITED SPEED BIT 0
   // SLS0  SLS1
   //    0        0   BA1 DOOR OPEN
   //    1        0   BA2
   //    0        1   BA3 SEMICYCLE WITH LOAD DOOR OPEN
   //    1        1   ALL DOOR CLOSED
   RUNG wire#powerrail
      Contact( "DB1018_SAFETY_TAGS".GROUP_9_C23_X23_Z23.SLS_BIT0 )
      wire#w1
      Coil( "C23_SAFETY_OUT".Select_SLS_bit_0 )
   END_RUNG
   RUNG wire#w1
      Coil( "X23_SAFETY_OUT".Select_SLS_bit_0 )
   END_RUNG
   RUNG wire#w1
      Coil( "Z23_SAFETY_OUT".Select_SLS_bit_0 )
   END_RUNG
   // the same network as SCL:
   "C23_SAFETY_OUT".Select_SLS_bit_0 := "DB1018_SAFETY_TAGS".GROUP_9_C23_X23_Z23.SLS_BIT0;
   "X23_SAFETY_OUT".Select_SLS_bit_0 := "DB1018_SAFETY_TAGS".GROUP_9_C23_X23_Z23.SLS_BIT0;
   "Z23_SAFETY_OUT".Select_SLS_bit_0 := "DB1018_SAFETY_TAGS".GROUP_9_C23_X23_Z23.SLS_BIT0;
END_REGION

REGION Network 201: GROUP 9 SAFE LIMITED SPEED BIT 1
   // SLS0  SLS1
   //    0        0   BA1 DOOR OPEN
   //    1        0   BA2
   //    0        1   BA3 SEMICYCLE WITH LOAD DOOR OPEN
   //    1        1   ALL DOOR CLOSED
   RUNG wire#powerrail
      Contact( "DB1018_SAFETY_TAGS".SAFE_DOORS_U02_CLOSED_AND_LOCKED )
      wire#w1
      Coil( "DB1018_SAFETY_TAGS".GROUP_9_C23_X23_Z23.SLS_BIT1 )
   END_RUNG
   RUNG wire#powerrail
      Contact( "DB2001_MODES_GENERAL".BA.BA3_SELECTED )
      Contact( "DB1018_SAFETY_TAGS".POWER_ON_W_ENABLE_BUTT )
   END_RUNG wire#w1
   // the same network as SCL:
   "DB1018_SAFETY_TAGS".GROUP_9_C23_X23_Z23.SLS_BIT1 := "DB1018_SAFETY_TAGS".SAFE_DOORS_U02_CLOSED_AND_LOCKED OR ("DB2001_MODES_GENERAL".BA.BA3_SELECTED AND "DB1018_SAFETY_TAGS".POWER_ON_W_ENABLE_BUTT);
END_REGION

REGION Network 202: SELECT SAFE LIMITED SPEED BIT 1
   // SLS0  SLS1
   //    0        0   BA1 DOOR OPEN
   //    1        0   BA2
   //    0        1   BA3 SEMICYCLE WITH LOAD DOOR OPEN
   //    1        1   ALL DOOR CLOSED
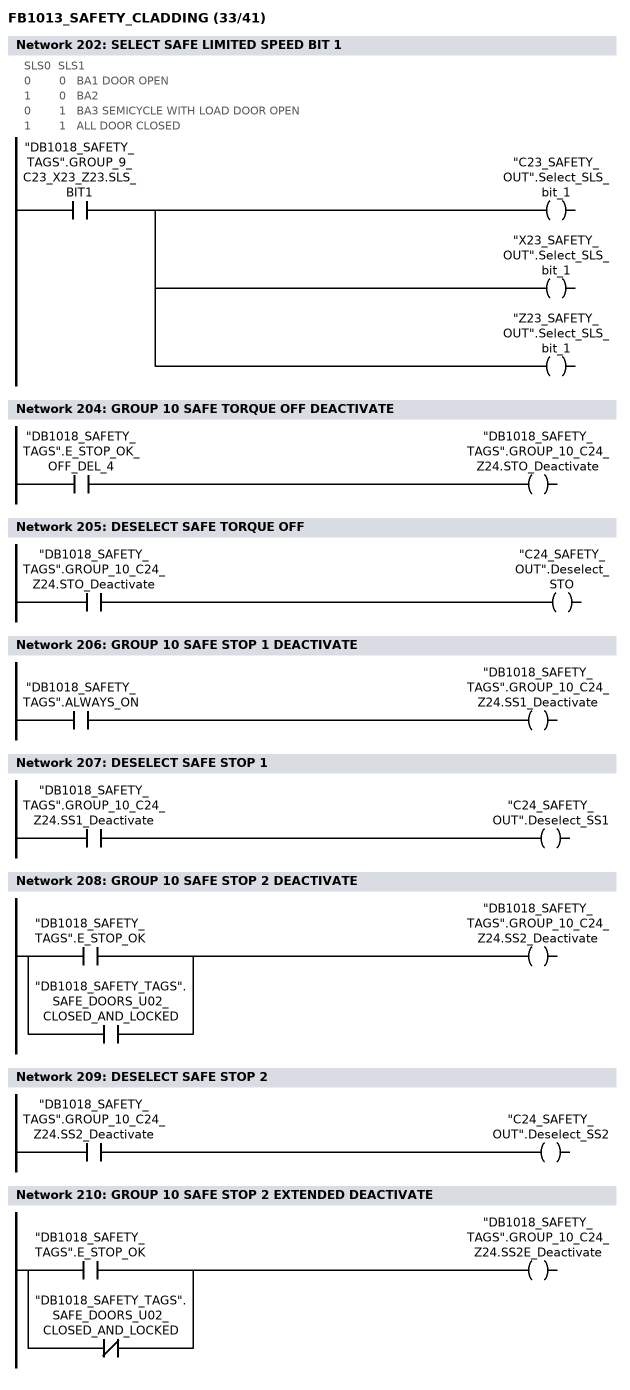
   RUNG wire#powerrail
      Contact( "DB1018_SAFETY_TAGS".GROUP_9_C23_X23_Z23.SLS_BIT1 )
      wire#w1
      Coil( "C23_SAFETY_OUT".Select_SLS_bit_1 )
   END_RUNG
   RUNG wire#w1
      Coil( "X23_SAFETY_OUT".Select_SLS_bit_1 )
   END_RUNG
   RUNG wire#w1
      Coil( "Z23_SAFETY_OUT".Select_SLS_bit_1 )
   END_RUNG
   // the same network as SCL:
   "C23_SAFETY_OUT".Select_SLS_bit_1 := "DB1018_SAFETY_TAGS".GROUP_9_C23_X23_Z23.SLS_BIT1;
   "X23_SAFETY_OUT".Select_SLS_bit_1 := "DB1018_SAFETY_TAGS".GROUP_9_C23_X23_Z23.SLS_BIT1;
   "Z23_SAFETY_OUT".Select_SLS_bit_1 := "DB1018_SAFETY_TAGS".GROUP_9_C23_X23_Z23.SLS_BIT1;
END_REGION

REGION Network 203: *************** GROUP 10 - C24 ***************
END_REGION

REGION Network 204: GROUP 10 SAFE TORQUE OFF DEACTIVATE
   RUNG wire#powerrail
      Contact( "DB1018_SAFETY_TAGS".E_STOP_OK_OFF_DEL_4 )
      Coil( "DB1018_SAFETY_TAGS".GROUP_10_C24_Z24.STO_Deactivate )
   END_RUNG
   // the same network as SCL:
   "DB1018_SAFETY_TAGS".GROUP_10_C24_Z24.STO_Deactivate := "DB1018_SAFETY_TAGS".E_STOP_OK_OFF_DEL_4;
END_REGION

REGION Network 205: DESELECT SAFE TORQUE OFF
   RUNG wire#powerrail
      Contact( "DB1018_SAFETY_TAGS".GROUP_10_C24_Z24.STO_Deactivate )
      Coil( "C24_SAFETY_OUT".Deselect_STO )
   END_RUNG
   // the same network as SCL:
   "C24_SAFETY_OUT".Deselect_STO := "DB1018_SAFETY_TAGS".GROUP_10_C24_Z24.STO_Deactivate;
END_REGION

REGION Network 206: GROUP 10 SAFE STOP 1 DEACTIVATE
   RUNG wire#powerrail
      Contact( "DB1018_SAFETY_TAGS".ALWAYS_ON )
      Coil( "DB1018_SAFETY_TAGS".GROUP_10_C24_Z24.SS1_Deactivate )
   END_RUNG
   // the same network as SCL:
   "DB1018_SAFETY_TAGS".GROUP_10_C24_Z24.SS1_Deactivate := "DB1018_SAFETY_TAGS".ALWAYS_ON;
END_REGION

REGION Network 207: DESELECT SAFE STOP 1
   RUNG wire#powerrail
      Contact( "DB1018_SAFETY_TAGS".GROUP_10_C24_Z24.SS1_Deactivate )
      Coil( "C24_SAFETY_OUT".Deselect_SS1 )
   END_RUNG
   // the same network as SCL:
   "C24_SAFETY_OUT".Deselect_SS1 := "DB1018_SAFETY_TAGS".GROUP_10_C24_Z24.SS1_Deactivate;
END_REGION

REGION Network 208: GROUP 10 SAFE STOP 2 DEACTIVATE
   RUNG wire#powerrail
      Contact( "DB1018_SAFETY_TAGS".E_STOP_OK )
      wire#w1
      Coil( "DB1018_SAFETY_TAGS".GROUP_10_C24_Z24.SS2_Deactivate )
   END_RUNG
   RUNG wire#powerrail
      Contact( "DB1018_SAFETY_TAGS".SAFE_DOORS_U02_CLOSED_AND_LOCKED )
   END_RUNG wire#w1
   // the same network as SCL:
   "DB1018_SAFETY_TAGS".GROUP_10_C24_Z24.SS2_Deactivate := "DB1018_SAFETY_TAGS".E_STOP_OK OR "DB1018_SAFETY_TAGS".SAFE_DOORS_U02_CLOSED_AND_LOCKED;
END_REGION

REGION Network 209: DESELECT SAFE STOP 2
   RUNG wire#powerrail
      Contact( "DB1018_SAFETY_TAGS".GROUP_10_C24_Z24.SS2_Deactivate )
      Coil( "C24_SAFETY_OUT".Deselect_SS2 )
   END_RUNG
   // the same network as SCL:
   "C24_SAFETY_OUT".Deselect_SS2 := "DB1018_SAFETY_TAGS".GROUP_10_C24_Z24.SS2_Deactivate;
END_REGION

REGION Network 210: GROUP 10 SAFE STOP 2 EXTENDED DEACTIVATE
   RUNG wire#powerrail
      Contact( "DB1018_SAFETY_TAGS".E_STOP_OK )
      wire#w1
      Coil( "DB1018_SAFETY_TAGS".GROUP_10_C24_Z24.SS2E_Deactivate )
   END_RUNG
   RUNG wire#powerrail
      I_Contact( "DB1018_SAFETY_TAGS".SAFE_DOORS_U02_CLOSED_AND_LOCKED )
   END_RUNG wire#w1
   // the same network as SCL:
   "DB1018_SAFETY_TAGS".GROUP_10_C24_Z24.SS2E_Deactivate := "DB1018_SAFETY_TAGS".E_STOP_OK OR NOT "DB1018_SAFETY_TAGS".SAFE_DOORS_U02_CLOSED_AND_LOCKED;
END_REGION

REGION Network 211: DESELECT SAFE STOP 2 EXTENDED
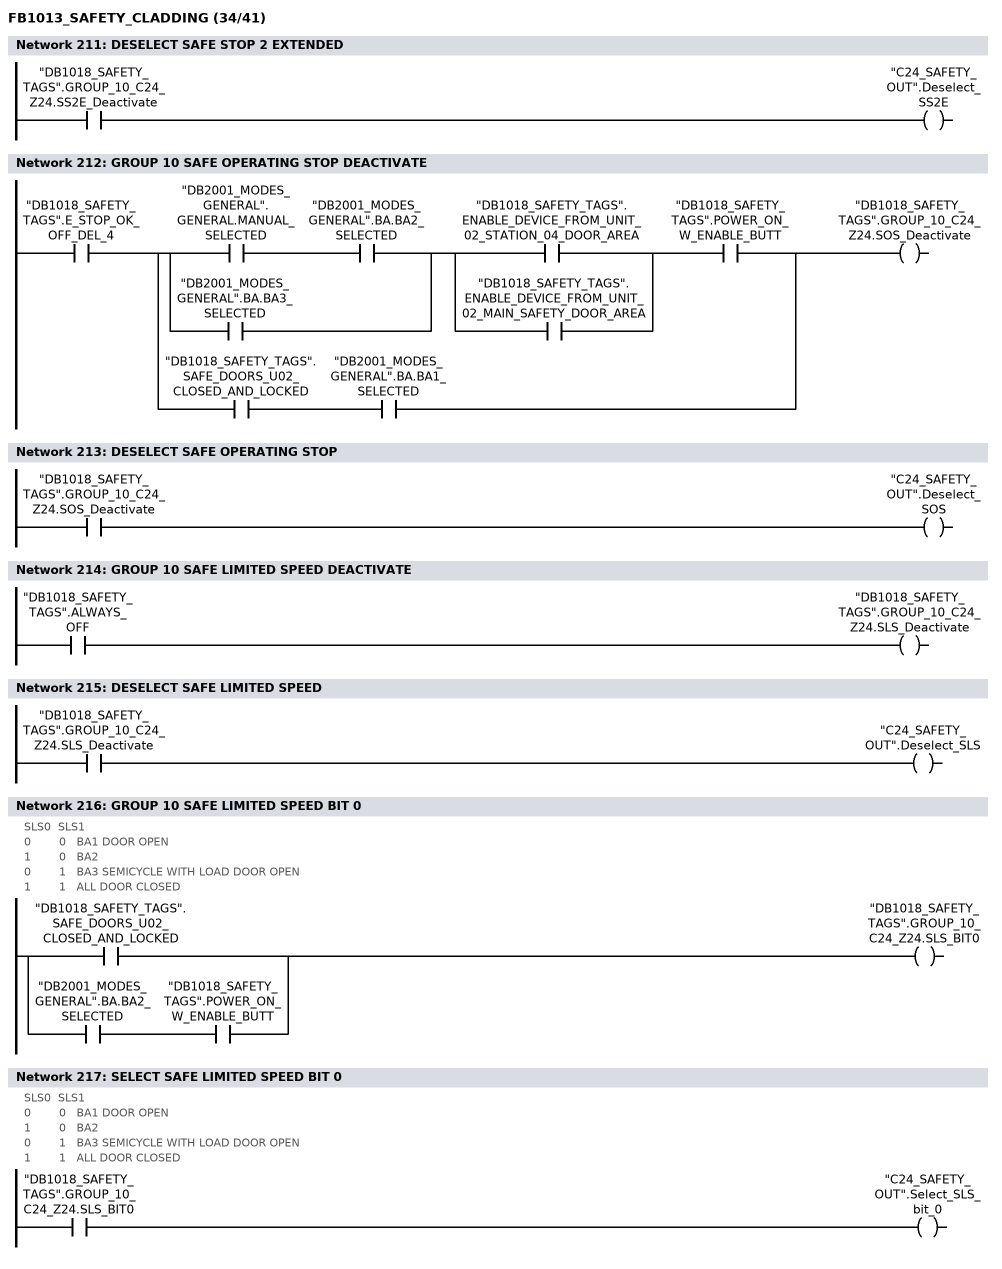
   RUNG wire#powerrail
      Contact( "DB1018_SAFETY_TAGS".GROUP_10_C24_Z24.SS2E_Deactivate )
      Coil( "C24_SAFETY_OUT".Deselect_SS2E )
   END_RUNG
   // the same network as SCL:
   "C24_SAFETY_OUT".Deselect_SS2E := "DB1018_SAFETY_TAGS".GROUP_10_C24_Z24.SS2E_Deactivate;
END_REGION

REGION Network 212: GROUP 10 SAFE OPERATING STOP DEACTIVATE
   RUNG wire#powerrail
      Contact( "DB1018_SAFETY_TAGS".E_STOP_OK_OFF_DEL_4 )
      wire#w1
      Contact( "DB2001_MODES_GENERAL".GENERAL.MANUAL_SELECTED )
      Contact( "DB2001_MODES_GENERAL".BA.BA2_SELECTED )
      wire#w2
      Contact( "DB1018_SAFETY_TAGS".ENABLE_DEVICE_FROM_UNIT_02_STATION_04_DOOR_AREA )
      wire#w3
      Contact( "DB1018_SAFETY_TAGS".POWER_ON_W_ENABLE_BUTT )
      wire#w4
      Coil( "DB1018_SAFETY_TAGS".GROUP_10_C24_Z24.SOS_Deactivate )
   END_RUNG
   RUNG wire#w1
      Contact( "DB2001_MODES_GENERAL".BA.BA3_SELECTED )
   END_RUNG wire#w2
   RUNG wire#w2
      Contact( "DB1018_SAFETY_TAGS".ENABLE_DEVICE_FROM_UNIT_02_MAIN_SAFETY_DOOR_AREA )
   END_RUNG wire#w3
   RUNG wire#w1
      Contact( "DB1018_SAFETY_TAGS".SAFE_DOORS_U02_CLOSED_AND_LOCKED )
      Contact( "DB2001_MODES_GENERAL".BA.BA1_SELECTED )
   END_RUNG wire#w4
   // the same network as SCL:
   "DB1018_SAFETY_TAGS".GROUP_10_C24_Z24.SOS_Deactivate := "DB1018_SAFETY_TAGS".E_STOP_OK_OFF_DEL_4 AND (((("DB2001_MODES_GENERAL".GENERAL.MANUAL_SELECTED AND "DB2001_MODES_GENERAL".BA.BA2_SELECTED) OR "DB2001_MODES_GENERAL".BA.BA3_SELECTED) AND ("DB1018_SAFETY_TAGS".ENABLE_DEVICE_FROM_UNIT_02_STATION_04_DOOR_AREA OR "DB1018_SAFETY_TAGS".ENABLE_DEVICE_FROM_UNIT_02_MAIN_SAFETY_DOOR_AREA) AND "DB1018_SAFETY_TAGS".POWER_ON_W_ENABLE_BUTT) OR ("DB1018_SAFETY_TAGS".SAFE_DOORS_U02_CLOSED_AND_LOCKED AND "DB2001_MODES_GENERAL".BA.BA1_SELECTED));
END_REGION

REGION Network 213: DESELECT SAFE OPERATING STOP
   RUNG wire#powerrail
      Contact( "DB1018_SAFETY_TAGS".GROUP_10_C24_Z24.SOS_Deactivate )
      Coil( "C24_SAFETY_OUT".Deselect_SOS )
   END_RUNG
   // the same network as SCL:
   "C24_SAFETY_OUT".Deselect_SOS := "DB1018_SAFETY_TAGS".GROUP_10_C24_Z24.SOS_Deactivate;
END_REGION

REGION Network 214: GROUP 10 SAFE LIMITED SPEED DEACTIVATE
   RUNG wire#powerrail
      Contact( "DB1018_SAFETY_TAGS".ALWAYS_OFF )
      Coil( "DB1018_SAFETY_TAGS".GROUP_10_C24_Z24.SLS_Deactivate )
   END_RUNG
   // the same network as SCL:
   "DB1018_SAFETY_TAGS".GROUP_10_C24_Z24.SLS_Deactivate := "DB1018_SAFETY_TAGS".ALWAYS_OFF;
END_REGION

REGION Network 215: DESELECT SAFE LIMITED SPEED
   RUNG wire#powerrail
      Contact( "DB1018_SAFETY_TAGS".GROUP_10_C24_Z24.SLS_Deactivate )
      Coil( "C24_SAFETY_OUT".Deselect_SLS )
   END_RUNG
   // the same network as SCL:
   "C24_SAFETY_OUT".Deselect_SLS := "DB1018_SAFETY_TAGS".GROUP_10_C24_Z24.SLS_Deactivate;
END_REGION

REGION Network 216: GROUP 10 SAFE LIMITED SPEED BIT 0
   // SLS0  SLS1
   //    0        0   BA1 DOOR OPEN
   //    1        0   BA2
   //    0        1   BA3 SEMICYCLE WITH LOAD DOOR OPEN
   //    1        1   ALL DOOR CLOSED
   RUNG wire#powerrail
      Contact( "DB1018_SAFETY_TAGS".SAFE_DOORS_U02_CLOSED_AND_LOCKED )
      wire#w1
      Coil( "DB1018_SAFETY_TAGS".GROUP_10_C24_Z24.SLS_BIT0 )
   END_RUNG
   RUNG wire#powerrail
      Contact( "DB2001_MODES_GENERAL".BA.BA2_SELECTED )
      Contact( "DB1018_SAFETY_TAGS".POWER_ON_W_ENABLE_BUTT )
   END_RUNG wire#w1
   // the same network as SCL:
   "DB1018_SAFETY_TAGS".GROUP_10_C24_Z24.SLS_BIT0 := "DB1018_SAFETY_TAGS".SAFE_DOORS_U02_CLOSED_AND_LOCKED OR ("DB2001_MODES_GENERAL".BA.BA2_SELECTED AND "DB1018_SAFETY_TAGS".POWER_ON_W_ENABLE_BUTT);
END_REGION

REGION Network 217: SELECT SAFE LIMITED SPEED BIT 0
   // SLS0  SLS1
   //    0        0   BA1 DOOR OPEN
   //    1        0   BA2
   //    0        1   BA3 SEMICYCLE WITH LOAD DOOR OPEN
   //    1        1   ALL DOOR CLOSED
   RUNG wire#powerrail
      Contact( "DB1018_SAFETY_TAGS".GROUP_10_C24_Z24.SLS_BIT0 )
      Coil( "C24_SAFETY_OUT".Select_SLS_bit_0 )
   END_RUNG
   // the same network as SCL:
   "C24_SAFETY_OUT".Select_SLS_bit_0 := "DB1018_SAFETY_TAGS".GROUP_10_C24_Z24.SLS_BIT0;
END_REGION

REGION Network 218: GROUP 10 SAFE LIMITED SPEED BIT 1
   // SLS0  SLS1
   //    0        0   BA1 DOOR OPEN
   //    1        0   BA2
   //    0        1   BA3 SEMICYCLE WITH LOAD DOOR OPEN
   //    1        1   ALL DOOR CLOSED
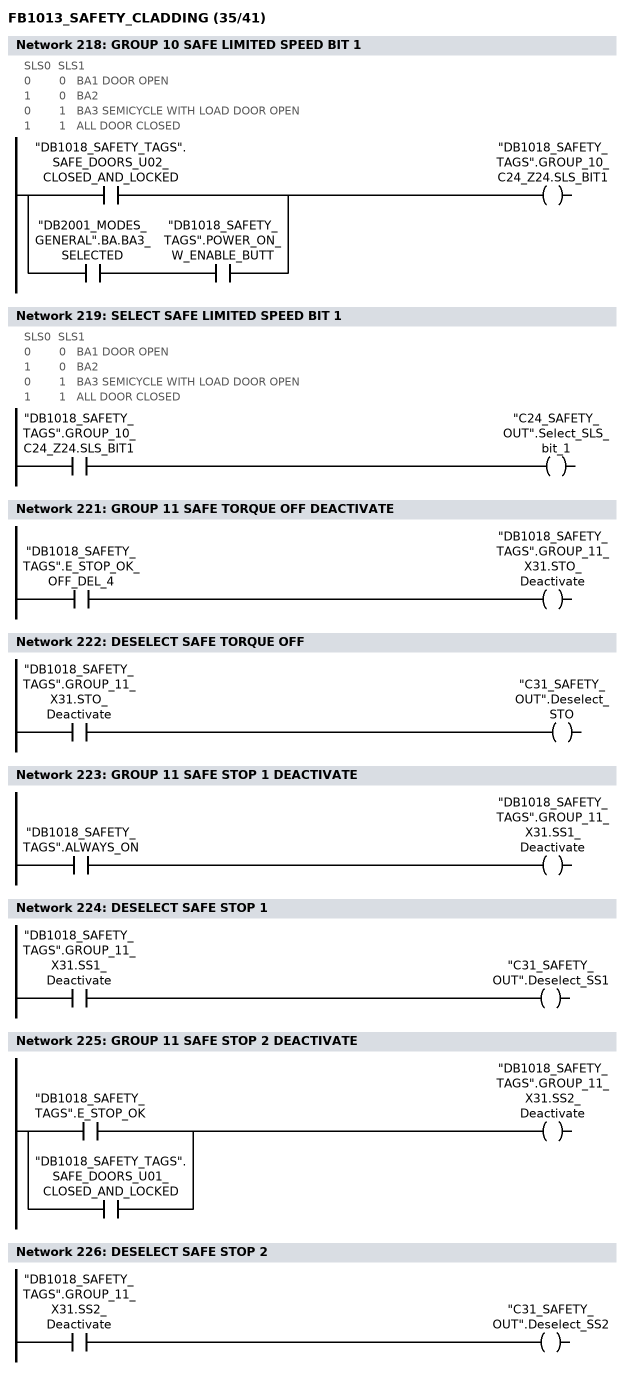
   RUNG wire#powerrail
      Contact( "DB1018_SAFETY_TAGS".SAFE_DOORS_U02_CLOSED_AND_LOCKED )
      wire#w1
      Coil( "DB1018_SAFETY_TAGS".GROUP_10_C24_Z24.SLS_BIT1 )
   END_RUNG
   RUNG wire#powerrail
      Contact( "DB2001_MODES_GENERAL".BA.BA3_SELECTED )
      Contact( "DB1018_SAFETY_TAGS".POWER_ON_W_ENABLE_BUTT )
   END_RUNG wire#w1
   // the same network as SCL:
   "DB1018_SAFETY_TAGS".GROUP_10_C24_Z24.SLS_BIT1 := "DB1018_SAFETY_TAGS".SAFE_DOORS_U02_CLOSED_AND_LOCKED OR ("DB2001_MODES_GENERAL".BA.BA3_SELECTED AND "DB1018_SAFETY_TAGS".POWER_ON_W_ENABLE_BUTT);
END_REGION

REGION Network 219: SELECT SAFE LIMITED SPEED BIT 1
   // SLS0  SLS1
   //    0        0   BA1 DOOR OPEN
   //    1        0   BA2
   //    0        1   BA3 SEMICYCLE WITH LOAD DOOR OPEN
   //    1        1   ALL DOOR CLOSED
   RUNG wire#powerrail
      Contact( "DB1018_SAFETY_TAGS".GROUP_10_C24_Z24.SLS_BIT1 )
      Coil( "C24_SAFETY_OUT".Select_SLS_bit_1 )
   END_RUNG
   // the same network as SCL:
   "C24_SAFETY_OUT".Select_SLS_bit_1 := "DB1018_SAFETY_TAGS".GROUP_10_C24_Z24.SLS_BIT1;
END_REGION

REGION Network 220: *************** GROUP 11 - C31 ***************
END_REGION

REGION Network 221: GROUP 11 SAFE TORQUE OFF DEACTIVATE
   RUNG wire#powerrail
      Contact( "DB1018_SAFETY_TAGS".E_STOP_OK_OFF_DEL_4 )
      Coil( "DB1018_SAFETY_TAGS".GROUP_11_X31.STO_Deactivate )
   END_RUNG
   // the same network as SCL:
   "DB1018_SAFETY_TAGS".GROUP_11_X31.STO_Deactivate := "DB1018_SAFETY_TAGS".E_STOP_OK_OFF_DEL_4;
END_REGION

REGION Network 222: DESELECT SAFE TORQUE OFF
   RUNG wire#powerrail
      Contact( "DB1018_SAFETY_TAGS".GROUP_11_X31.STO_Deactivate )
      Coil( "C31_SAFETY_OUT".Deselect_STO )
   END_RUNG
   // the same network as SCL:
   "C31_SAFETY_OUT".Deselect_STO := "DB1018_SAFETY_TAGS".GROUP_11_X31.STO_Deactivate;
END_REGION

REGION Network 223: GROUP 11 SAFE STOP 1 DEACTIVATE
   RUNG wire#powerrail
      Contact( "DB1018_SAFETY_TAGS".ALWAYS_ON )
      Coil( "DB1018_SAFETY_TAGS".GROUP_11_X31.SS1_Deactivate )
   END_RUNG
   // the same network as SCL:
   "DB1018_SAFETY_TAGS".GROUP_11_X31.SS1_Deactivate := "DB1018_SAFETY_TAGS".ALWAYS_ON;
END_REGION

REGION Network 224: DESELECT SAFE STOP 1
   RUNG wire#powerrail
      Contact( "DB1018_SAFETY_TAGS".GROUP_11_X31.SS1_Deactivate )
      Coil( "C31_SAFETY_OUT".Deselect_SS1 )
   END_RUNG
   // the same network as SCL:
   "C31_SAFETY_OUT".Deselect_SS1 := "DB1018_SAFETY_TAGS".GROUP_11_X31.SS1_Deactivate;
END_REGION

REGION Network 225: GROUP 11 SAFE STOP 2 DEACTIVATE
   RUNG wire#powerrail
      Contact( "DB1018_SAFETY_TAGS".E_STOP_OK )
      wire#w1
      Coil( "DB1018_SAFETY_TAGS".GROUP_11_X31.SS2_Deactivate )
   END_RUNG
   RUNG wire#powerrail
      Contact( "DB1018_SAFETY_TAGS".SAFE_DOORS_U01_CLOSED_AND_LOCKED )
   END_RUNG wire#w1
   // the same network as SCL:
   "DB1018_SAFETY_TAGS".GROUP_11_X31.SS2_Deactivate := "DB1018_SAFETY_TAGS".E_STOP_OK OR "DB1018_SAFETY_TAGS".SAFE_DOORS_U01_CLOSED_AND_LOCKED;
END_REGION

REGION Network 226: DESELECT SAFE STOP 2
   RUNG wire#powerrail
      Contact( "DB1018_SAFETY_TAGS".GROUP_11_X31.SS2_Deactivate )
      Coil( "C31_SAFETY_OUT".Deselect_SS2 )
   END_RUNG
   // the same network as SCL:
   "C31_SAFETY_OUT".Deselect_SS2 := "DB1018_SAFETY_TAGS".GROUP_11_X31.SS2_Deactivate;
END_REGION

REGION Network 227: GROUP 11 SAFE STOP 2 EXTENDED DEACTIVATE
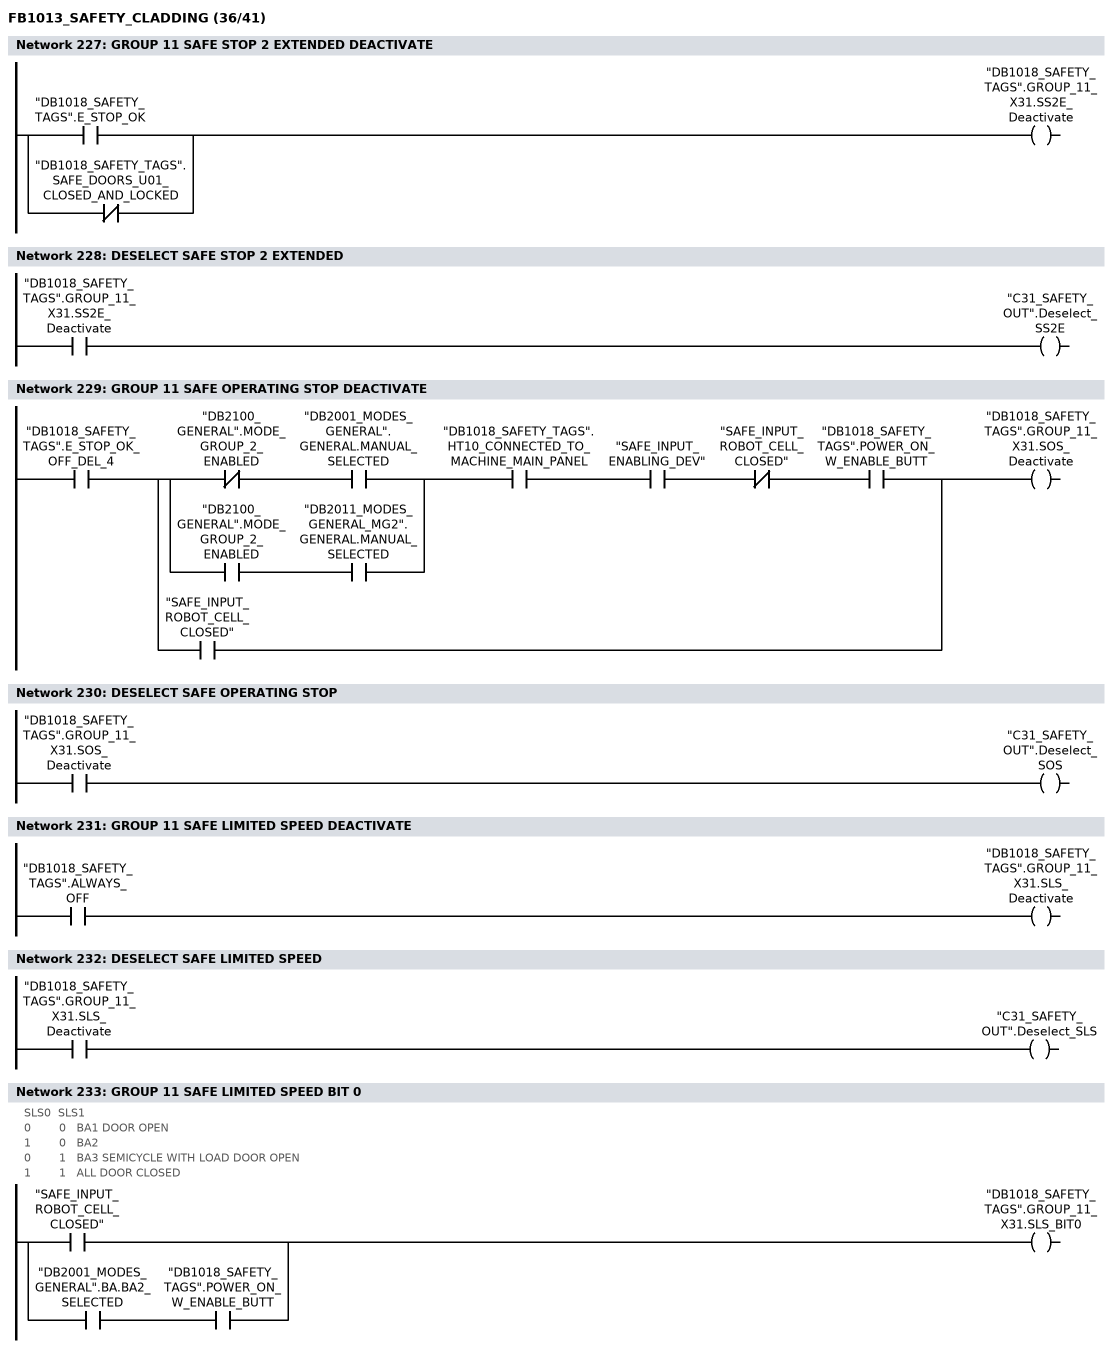
   RUNG wire#powerrail
      Contact( "DB1018_SAFETY_TAGS".E_STOP_OK )
      wire#w1
      Coil( "DB1018_SAFETY_TAGS".GROUP_11_X31.SS2E_Deactivate )
   END_RUNG
   RUNG wire#powerrail
      I_Contact( "DB1018_SAFETY_TAGS".SAFE_DOORS_U01_CLOSED_AND_LOCKED )
   END_RUNG wire#w1
   // the same network as SCL:
   "DB1018_SAFETY_TAGS".GROUP_11_X31.SS2E_Deactivate := "DB1018_SAFETY_TAGS".E_STOP_OK OR NOT "DB1018_SAFETY_TAGS".SAFE_DOORS_U01_CLOSED_AND_LOCKED;
END_REGION

REGION Network 228: DESELECT SAFE STOP 2 EXTENDED
   RUNG wire#powerrail
      Contact( "DB1018_SAFETY_TAGS".GROUP_11_X31.SS2E_Deactivate )
      Coil( "C31_SAFETY_OUT".Deselect_SS2E )
   END_RUNG
   // the same network as SCL:
   "C31_SAFETY_OUT".Deselect_SS2E := "DB1018_SAFETY_TAGS".GROUP_11_X31.SS2E_Deactivate;
END_REGION

REGION Network 229: GROUP 11 SAFE OPERATING STOP DEACTIVATE
   RUNG wire#powerrail
      Contact( "DB1018_SAFETY_TAGS".E_STOP_OK_OFF_DEL_4 )
      wire#w1
      I_Contact( "DB2100_GENERAL".MODE_GROUP_2_ENABLED )
      Contact( "DB2001_MODES_GENERAL".GENERAL.MANUAL_SELECTED )
      wire#w2
      Contact( "DB1018_SAFETY_TAGS".HT10_CONNECTED_TO_MACHINE_MAIN_PANEL )
      Contact( "SAFE_INPUT_ENABLING_DEV" )
      I_Contact( "SAFE_INPUT_ROBOT_CELL_CLOSED" )
      Contact( "DB1018_SAFETY_TAGS".POWER_ON_W_ENABLE_BUTT )
      wire#w3
      Coil( "DB1018_SAFETY_TAGS".GROUP_11_X31.SOS_Deactivate )
   END_RUNG
   RUNG wire#w1
      Contact( "DB2100_GENERAL".MODE_GROUP_2_ENABLED )
      Contact( "DB2011_MODES_GENERAL_MG2".GENERAL.MANUAL_SELECTED )
   END_RUNG wire#w2
   RUNG wire#w1
      Contact( "SAFE_INPUT_ROBOT_CELL_CLOSED" )
   END_RUNG wire#w3
   // the same network as SCL:
   "DB1018_SAFETY_TAGS".GROUP_11_X31.SOS_Deactivate := "DB1018_SAFETY_TAGS".E_STOP_OK_OFF_DEL_4 AND ((((NOT "DB2100_GENERAL".MODE_GROUP_2_ENABLED AND "DB2001_MODES_GENERAL".GENERAL.MANUAL_SELECTED) OR ("DB2100_GENERAL".MODE_GROUP_2_ENABLED AND "DB2011_MODES_GENERAL_MG2".GENERAL.MANUAL_SELECTED)) AND "DB1018_SAFETY_TAGS".HT10_CONNECTED_TO_MACHINE_MAIN_PANEL AND "SAFE_INPUT_ENABLING_DEV" AND NOT "SAFE_INPUT_ROBOT_CELL_CLOSED" AND "DB1018_SAFETY_TAGS".POWER_ON_W_ENABLE_BUTT) OR "SAFE_INPUT_ROBOT_CELL_CLOSED");
END_REGION

REGION Network 230: DESELECT SAFE OPERATING STOP
   RUNG wire#powerrail
      Contact( "DB1018_SAFETY_TAGS".GROUP_11_X31.SOS_Deactivate )
      Coil( "C31_SAFETY_OUT".Deselect_SOS )
   END_RUNG
   // the same network as SCL:
   "C31_SAFETY_OUT".Deselect_SOS := "DB1018_SAFETY_TAGS".GROUP_11_X31.SOS_Deactivate;
END_REGION

REGION Network 231: GROUP 11 SAFE LIMITED SPEED DEACTIVATE
   RUNG wire#powerrail
      Contact( "DB1018_SAFETY_TAGS".ALWAYS_OFF )
      Coil( "DB1018_SAFETY_TAGS".GROUP_11_X31.SLS_Deactivate )
   END_RUNG
   // the same network as SCL:
   "DB1018_SAFETY_TAGS".GROUP_11_X31.SLS_Deactivate := "DB1018_SAFETY_TAGS".ALWAYS_OFF;
END_REGION

REGION Network 232: DESELECT SAFE LIMITED SPEED
   RUNG wire#powerrail
      Contact( "DB1018_SAFETY_TAGS".GROUP_11_X31.SLS_Deactivate )
      Coil( "C31_SAFETY_OUT".Deselect_SLS )
   END_RUNG
   // the same network as SCL:
   "C31_SAFETY_OUT".Deselect_SLS := "DB1018_SAFETY_TAGS".GROUP_11_X31.SLS_Deactivate;
END_REGION

REGION Network 233: GROUP 11 SAFE LIMITED SPEED BIT 0
   // SLS0  SLS1
   //    0        0   BA1 DOOR OPEN
   //    1        0   BA2
   //    0        1   BA3 SEMICYCLE WITH LOAD DOOR OPEN
   //    1        1   ALL DOOR CLOSED
   RUNG wire#powerrail
      Contact( "SAFE_INPUT_ROBOT_CELL_CLOSED" )
      wire#w1
      Coil( "DB1018_SAFETY_TAGS".GROUP_11_X31.SLS_BIT0 )
   END_RUNG
   RUNG wire#powerrail
      Contact( "DB2001_MODES_GENERAL".BA.BA2_SELECTED )
      Contact( "DB1018_SAFETY_TAGS".POWER_ON_W_ENABLE_BUTT )
   END_RUNG wire#w1
   // the same network as SCL:
   "DB1018_SAFETY_TAGS".GROUP_11_X31.SLS_BIT0 := "SAFE_INPUT_ROBOT_CELL_CLOSED" OR ("DB2001_MODES_GENERAL".BA.BA2_SELECTED AND "DB1018_SAFETY_TAGS".POWER_ON_W_ENABLE_BUTT);
END_REGION

REGION Network 234: SELECT SAFE LIMITED SPEED BIT 0
   // SLS0  SLS1
   //    0        0   BA1 DOOR OPEN
   //    1        0   BA2
   //    0        1   BA3 SEMICYCLE WITH LOAD DOOR OPEN
   //    1        1   ALL DOOR CLOSED
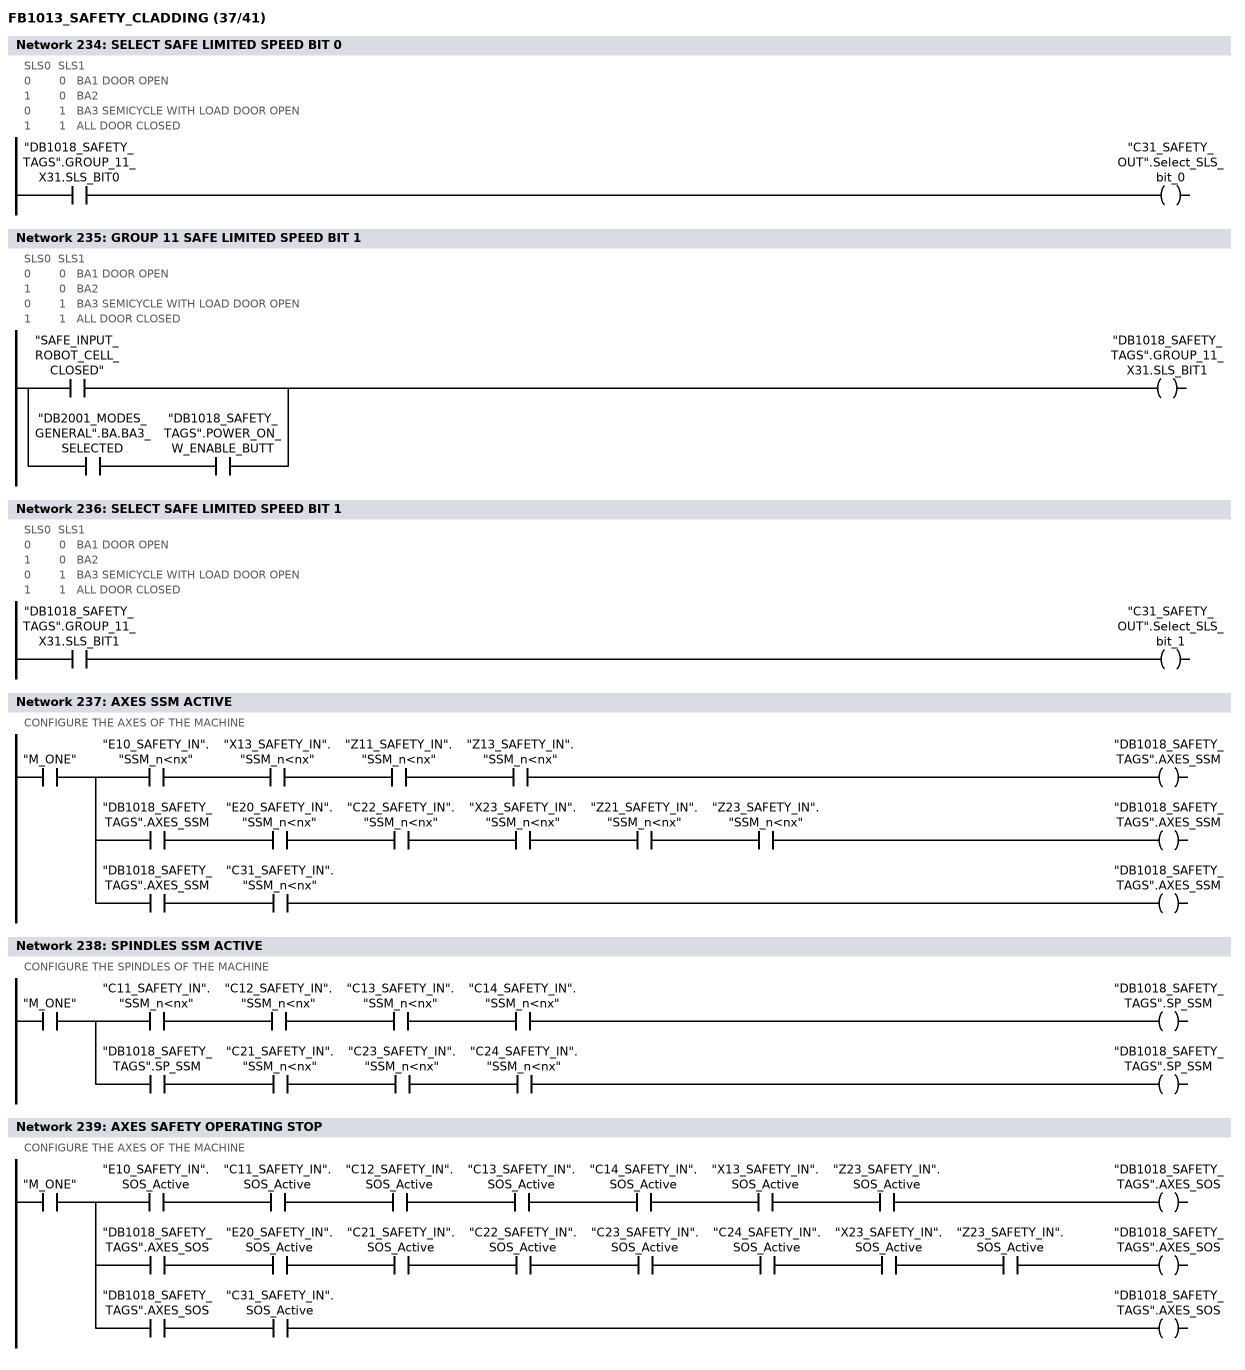
   RUNG wire#powerrail
      Contact( "DB1018_SAFETY_TAGS".GROUP_11_X31.SLS_BIT0 )
      Coil( "C31_SAFETY_OUT".Select_SLS_bit_0 )
   END_RUNG
   // the same network as SCL:
   "C31_SAFETY_OUT".Select_SLS_bit_0 := "DB1018_SAFETY_TAGS".GROUP_11_X31.SLS_BIT0;
END_REGION

REGION Network 235: GROUP 11 SAFE LIMITED SPEED BIT 1
   // SLS0  SLS1
   //    0        0   BA1 DOOR OPEN
   //    1        0   BA2
   //    0        1   BA3 SEMICYCLE WITH LOAD DOOR OPEN
   //    1        1   ALL DOOR CLOSED
   RUNG wire#powerrail
      Contact( "SAFE_INPUT_ROBOT_CELL_CLOSED" )
      wire#w1
      Coil( "DB1018_SAFETY_TAGS".GROUP_11_X31.SLS_BIT1 )
   END_RUNG
   RUNG wire#powerrail
      Contact( "DB2001_MODES_GENERAL".BA.BA3_SELECTED )
      Contact( "DB1018_SAFETY_TAGS".POWER_ON_W_ENABLE_BUTT )
   END_RUNG wire#w1
   // the same network as SCL:
   "DB1018_SAFETY_TAGS".GROUP_11_X31.SLS_BIT1 := "SAFE_INPUT_ROBOT_CELL_CLOSED" OR ("DB2001_MODES_GENERAL".BA.BA3_SELECTED AND "DB1018_SAFETY_TAGS".POWER_ON_W_ENABLE_BUTT);
END_REGION

REGION Network 236: SELECT SAFE LIMITED SPEED BIT 1
   // SLS0  SLS1
   //    0        0   BA1 DOOR OPEN
   //    1        0   BA2
   //    0        1   BA3 SEMICYCLE WITH LOAD DOOR OPEN
   //    1        1   ALL DOOR CLOSED
   RUNG wire#powerrail
      Contact( "DB1018_SAFETY_TAGS".GROUP_11_X31.SLS_BIT1 )
      Coil( "C31_SAFETY_OUT".Select_SLS_bit_1 )
   END_RUNG
   // the same network as SCL:
   "C31_SAFETY_OUT".Select_SLS_bit_1 := "DB1018_SAFETY_TAGS".GROUP_11_X31.SLS_BIT1;
END_REGION

REGION Network 237: AXES SSM ACTIVE
   // CONFIGURE THE AXES OF THE MACHINE
   RUNG wire#powerrail
      Contact( "M_ONE" )
      wire#w1
      Contact( "E10_SAFETY_IN"."SSM_n<nx" )
      Contact( "X13_SAFETY_IN"."SSM_n<nx" )
      Contact( "Z11_SAFETY_IN"."SSM_n<nx" )
      Contact( "Z13_SAFETY_IN"."SSM_n<nx" )
      Coil( "DB1018_SAFETY_TAGS".AXES_SSM )
   END_RUNG
   RUNG wire#w1
      Contact( "DB1018_SAFETY_TAGS".AXES_SSM )
      Contact( "E20_SAFETY_IN"."SSM_n<nx" )
      Contact( "C22_SAFETY_IN"."SSM_n<nx" )
      Contact( "X23_SAFETY_IN"."SSM_n<nx" )
      Contact( "Z21_SAFETY_IN"."SSM_n<nx" )
      Contact( "Z23_SAFETY_IN"."SSM_n<nx" )
      Coil( "DB1018_SAFETY_TAGS".AXES_SSM )
   END_RUNG
   RUNG wire#w1
      Contact( "DB1018_SAFETY_TAGS".AXES_SSM )
      Contact( "C31_SAFETY_IN"."SSM_n<nx" )
      Coil( "DB1018_SAFETY_TAGS".AXES_SSM )
   END_RUNG
   // the same network as SCL:
   "DB1018_SAFETY_TAGS".AXES_SSM := "M_ONE" AND "E10_SAFETY_IN"."SSM_n<nx" AND "X13_SAFETY_IN"."SSM_n<nx" AND "Z11_SAFETY_IN"."SSM_n<nx" AND "Z13_SAFETY_IN"."SSM_n<nx";
   "DB1018_SAFETY_TAGS".AXES_SSM := "M_ONE" AND "DB1018_SAFETY_TAGS".AXES_SSM AND "E20_SAFETY_IN"."SSM_n<nx" AND "C22_SAFETY_IN"."SSM_n<nx" AND "X23_SAFETY_IN"."SSM_n<nx" AND "Z21_SAFETY_IN"."SSM_n<nx" AND "Z23_SAFETY_IN"."SSM_n<nx";
   "DB1018_SAFETY_TAGS".AXES_SSM := "M_ONE" AND "DB1018_SAFETY_TAGS".AXES_SSM AND "C31_SAFETY_IN"."SSM_n<nx";
END_REGION

REGION Network 238: SPINDLES SSM ACTIVE
   // CONFIGURE THE SPINDLES OF THE MACHINE
   RUNG wire#powerrail
      Contact( "M_ONE" )
      wire#w1
      Contact( "C11_SAFETY_IN"."SSM_n<nx" )
      Contact( "C12_SAFETY_IN"."SSM_n<nx" )
      Contact( "C13_SAFETY_IN"."SSM_n<nx" )
      Contact( "C14_SAFETY_IN"."SSM_n<nx" )
      Coil( "DB1018_SAFETY_TAGS".SP_SSM )
   END_RUNG
   RUNG wire#w1
      Contact( "DB1018_SAFETY_TAGS".SP_SSM )
      Contact( "C21_SAFETY_IN"."SSM_n<nx" )
      Contact( "C23_SAFETY_IN"."SSM_n<nx" )
      Contact( "C24_SAFETY_IN"."SSM_n<nx" )
      Coil( "DB1018_SAFETY_TAGS".SP_SSM )
   END_RUNG
   // the same network as SCL:
   "DB1018_SAFETY_TAGS".SP_SSM := "M_ONE" AND "C11_SAFETY_IN"."SSM_n<nx" AND "C12_SAFETY_IN"."SSM_n<nx" AND "C13_SAFETY_IN"."SSM_n<nx" AND "C14_SAFETY_IN"."SSM_n<nx";
   "DB1018_SAFETY_TAGS".SP_SSM := "M_ONE" AND "DB1018_SAFETY_TAGS".SP_SSM AND "C21_SAFETY_IN"."SSM_n<nx" AND "C23_SAFETY_IN"."SSM_n<nx" AND "C24_SAFETY_IN"."SSM_n<nx";
END_REGION

REGION Network 239: AXES SAFETY OPERATING STOP
   // CONFIGURE THE AXES OF THE MACHINE
   RUNG wire#powerrail
      Contact( "M_ONE" )
      wire#w1
      Contact( "E10_SAFETY_IN".SOS_Active )
      Contact( "C11_SAFETY_IN".SOS_Active )
      Contact( "C12_SAFETY_IN".SOS_Active )
      Contact( "C13_SAFETY_IN".SOS_Active )
      Contact( "C14_SAFETY_IN".SOS_Active )
      Contact( "X13_SAFETY_IN".SOS_Active )
      Contact( "Z23_SAFETY_IN".SOS_Active )
      Coil( "DB1018_SAFETY_TAGS".AXES_SOS )
   END_RUNG
   RUNG wire#w1
      Contact( "DB1018_SAFETY_TAGS".AXES_SOS )
      Contact( "E20_SAFETY_IN".SOS_Active )
      Contact( "C21_SAFETY_IN".SOS_Active )
      Contact( "C22_SAFETY_IN".SOS_Active )
      Contact( "C23_SAFETY_IN".SOS_Active )
      Contact( "C24_SAFETY_IN".SOS_Active )
      Contact( "X23_SAFETY_IN".SOS_Active )
      Contact( "Z23_SAFETY_IN".SOS_Active )
      Coil( "DB1018_SAFETY_TAGS".AXES_SOS )
   END_RUNG
   RUNG wire#w1
      Contact( "DB1018_SAFETY_TAGS".AXES_SOS )
      Contact( "C31_SAFETY_IN".SOS_Active )
      Coil( "DB1018_SAFETY_TAGS".AXES_SOS )
   END_RUNG
   // the same network as SCL:
   "DB1018_SAFETY_TAGS".AXES_SOS := "M_ONE" AND "E10_SAFETY_IN".SOS_Active AND "C11_SAFETY_IN".SOS_Active AND "C12_SAFETY_IN".SOS_Active AND "C13_SAFETY_IN".SOS_Active AND "C14_SAFETY_IN".SOS_Active AND "X13_SAFETY_IN".SOS_Active AND "Z23_SAFETY_IN".SOS_Active;
   "DB1018_SAFETY_TAGS".AXES_SOS := "M_ONE" AND "DB1018_SAFETY_TAGS".AXES_SOS AND "E20_SAFETY_IN".SOS_Active AND "C21_SAFETY_IN".SOS_Active AND "C22_SAFETY_IN".SOS_Active AND "C23_SAFETY_IN".SOS_Active AND "C24_SAFETY_IN".SOS_Active AND "X23_SAFETY_IN".SOS_Active AND "Z23_SAFETY_IN".SOS_Active;
   "DB1018_SAFETY_TAGS".AXES_SOS := "M_ONE" AND "DB1018_SAFETY_TAGS".AXES_SOS AND "C31_SAFETY_IN".SOS_Active;
END_REGION

REGION Network 240: SPINDLES SAFETY OPERATING STOP
   // CONFIGURE THE SPINDLES OF THE MACHINE
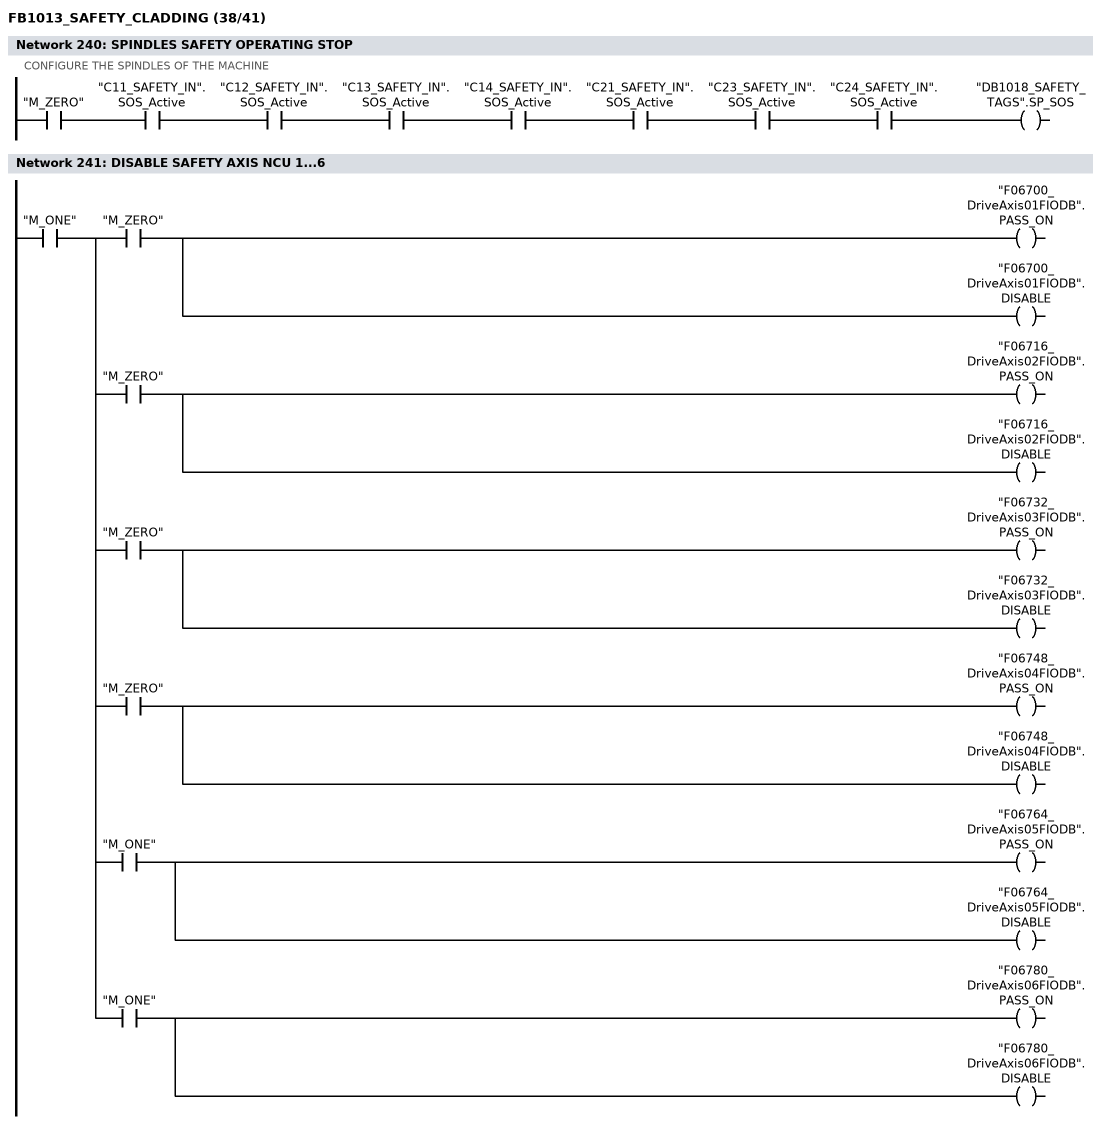
   RUNG wire#powerrail
      Contact( "M_ZERO" )
      Contact( "C11_SAFETY_IN".SOS_Active )
      Contact( "C12_SAFETY_IN".SOS_Active )
      Contact( "C13_SAFETY_IN".SOS_Active )
      Contact( "C14_SAFETY_IN".SOS_Active )
      Contact( "C21_SAFETY_IN".SOS_Active )
      Contact( "C23_SAFETY_IN".SOS_Active )
      Contact( "C24_SAFETY_IN".SOS_Active )
      Coil( "DB1018_SAFETY_TAGS".SP_SOS )
   END_RUNG
   // the same network as SCL:
   "DB1018_SAFETY_TAGS".SP_SOS := "M_ZERO" AND "C11_SAFETY_IN".SOS_Active AND "C12_SAFETY_IN".SOS_Active AND "C13_SAFETY_IN".SOS_Active AND "C14_SAFETY_IN".SOS_Active AND "C21_SAFETY_IN".SOS_Active AND "C23_SAFETY_IN".SOS_Active AND "C24_SAFETY_IN".SOS_Active;
END_REGION

REGION Network 241: DISABLE SAFETY AXIS NCU 1...6
   RUNG wire#powerrail
      Contact( "M_ONE" )
      wire#w1
      Contact( "M_ZERO" )
      wire#w2
      Coil( "F06700_DriveAxis01FIODB".PASS_ON )
   END_RUNG
   RUNG wire#w2
      Coil( "F06700_DriveAxis01FIODB".DISABLE )
   END_RUNG
   RUNG wire#w1
      Contact( "M_ZERO" )
      wire#w3
      Coil( "F06716_DriveAxis02FIODB".PASS_ON )
   END_RUNG
   RUNG wire#w3
      Coil( "F06716_DriveAxis02FIODB".DISABLE )
   END_RUNG
   RUNG wire#w1
      Contact( "M_ZERO" )
      wire#w4
      Coil( "F06732_DriveAxis03FIODB".PASS_ON )
   END_RUNG
   RUNG wire#w4
      Coil( "F06732_DriveAxis03FIODB".DISABLE )
   END_RUNG
   RUNG wire#w1
      Contact( "M_ZERO" )
      wire#w5
      Coil( "F06748_DriveAxis04FIODB".PASS_ON )
   END_RUNG
   RUNG wire#w5
      Coil( "F06748_DriveAxis04FIODB".DISABLE )
   END_RUNG
   RUNG wire#w1
      Contact( "M_ONE" )
      wire#w6
      Coil( "F06764_DriveAxis05FIODB".PASS_ON )
   END_RUNG
   RUNG wire#w6
      Coil( "F06764_DriveAxis05FIODB".DISABLE )
   END_RUNG
   RUNG wire#w1
      Contact( "M_ONE" )
      wire#w7
      Coil( "F06780_DriveAxis06FIODB".PASS_ON )
   END_RUNG
   RUNG wire#w7
      Coil( "F06780_DriveAxis06FIODB".DISABLE )
   END_RUNG
   // the same network as SCL:
   "F06700_DriveAxis01FIODB".PASS_ON := "M_ONE" AND "M_ZERO";
   "F06700_DriveAxis01FIODB".DISABLE := "F06700_DriveAxis01FIODB".PASS_ON;
   "F06716_DriveAxis02FIODB".PASS_ON := "M_ONE" AND "M_ZERO";
   "F06716_DriveAxis02FIODB".DISABLE := "F06716_DriveAxis02FIODB".PASS_ON;
   "F06732_DriveAxis03FIODB".PASS_ON := "M_ONE" AND "M_ZERO";
   "F06732_DriveAxis03FIODB".DISABLE := "F06732_DriveAxis03FIODB".PASS_ON;
   "F06748_DriveAxis04FIODB".PASS_ON := "M_ONE" AND "M_ZERO";
   "F06748_DriveAxis04FIODB".DISABLE := "F06748_DriveAxis04FIODB".PASS_ON;
   "F06764_DriveAxis05FIODB".PASS_ON := "M_ONE" AND "M_ONE";
   "F06764_DriveAxis05FIODB".DISABLE := "F06764_DriveAxis05FIODB".PASS_ON;
   "F06780_DriveAxis06FIODB".PASS_ON := "M_ONE" AND "M_ONE";
   "F06780_DriveAxis06FIODB".DISABLE := "F06780_DriveAxis06FIODB".PASS_ON;
END_REGION

REGION Network 242: DISABLE SAFETY AXIS NX15 7 ....12
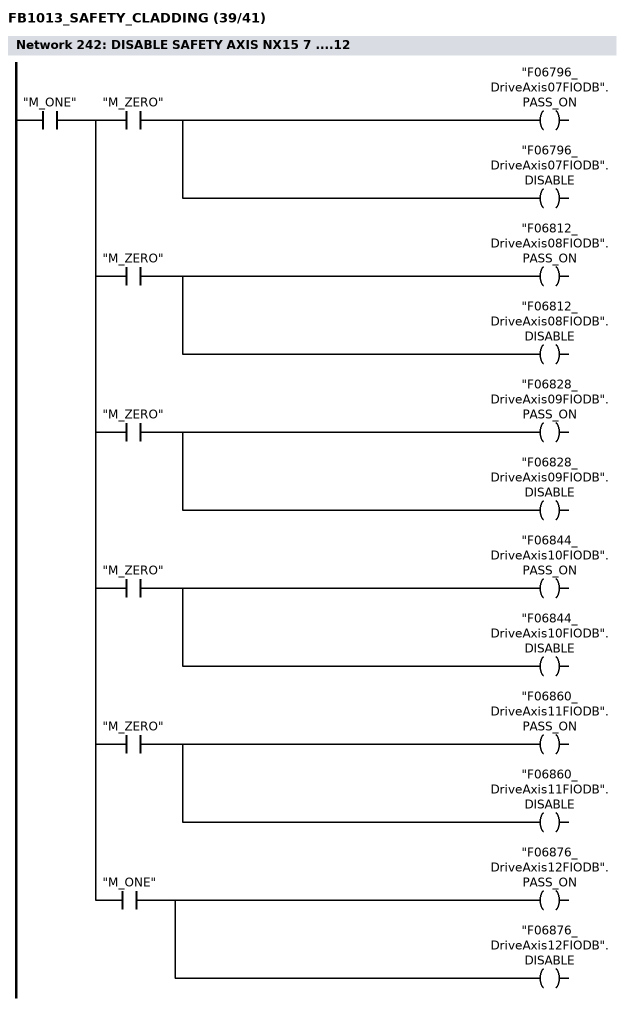
   RUNG wire#powerrail
      Contact( "M_ONE" )
      wire#w1
      Contact( "M_ZERO" )
      wire#w2
      Coil( "F06796_DriveAxis07FIODB".PASS_ON )
   END_RUNG
   RUNG wire#w2
      Coil( "F06796_DriveAxis07FIODB".DISABLE )
   END_RUNG
   RUNG wire#w1
      Contact( "M_ZERO" )
      wire#w3
      Coil( "F06812_DriveAxis08FIODB".PASS_ON )
   END_RUNG
   RUNG wire#w3
      Coil( "F06812_DriveAxis08FIODB".DISABLE )
   END_RUNG
   RUNG wire#w1
      Contact( "M_ZERO" )
      wire#w4
      Coil( "F06828_DriveAxis09FIODB".PASS_ON )
   END_RUNG
   RUNG wire#w4
      Coil( "F06828_DriveAxis09FIODB".DISABLE )
   END_RUNG
   RUNG wire#w1
      Contact( "M_ZERO" )
      wire#w5
      Coil( "F06844_DriveAxis10FIODB".PASS_ON )
   END_RUNG
   RUNG wire#w5
      Coil( "F06844_DriveAxis10FIODB".DISABLE )
   END_RUNG
   RUNG wire#w1
      Contact( "M_ZERO" )
      wire#w6
      Coil( "F06860_DriveAxis11FIODB".PASS_ON )
   END_RUNG
   RUNG wire#w6
      Coil( "F06860_DriveAxis11FIODB".DISABLE )
   END_RUNG
   RUNG wire#w1
      Contact( "M_ONE" )
      wire#w7
      Coil( "F06876_DriveAxis12FIODB".PASS_ON )
   END_RUNG
   RUNG wire#w7
      Coil( "F06876_DriveAxis12FIODB".DISABLE )
   END_RUNG
   // the same network as SCL:
   "F06796_DriveAxis07FIODB".PASS_ON := "M_ONE" AND "M_ZERO";
   "F06796_DriveAxis07FIODB".DISABLE := "F06796_DriveAxis07FIODB".PASS_ON;
   "F06812_DriveAxis08FIODB".PASS_ON := "M_ONE" AND "M_ZERO";
   "F06812_DriveAxis08FIODB".DISABLE := "F06812_DriveAxis08FIODB".PASS_ON;
   "F06828_DriveAxis09FIODB".PASS_ON := "M_ONE" AND "M_ZERO";
   "F06828_DriveAxis09FIODB".DISABLE := "F06828_DriveAxis09FIODB".PASS_ON;
   "F06844_DriveAxis10FIODB".PASS_ON := "M_ONE" AND "M_ZERO";
   "F06844_DriveAxis10FIODB".DISABLE := "F06844_DriveAxis10FIODB".PASS_ON;
   "F06860_DriveAxis11FIODB".PASS_ON := "M_ONE" AND "M_ZERO";
   "F06860_DriveAxis11FIODB".DISABLE := "F06860_DriveAxis11FIODB".PASS_ON;
   "F06876_DriveAxis12FIODB".PASS_ON := "M_ONE" AND "M_ONE";
   "F06876_DriveAxis12FIODB".DISABLE := "F06876_DriveAxis12FIODB".PASS_ON;
END_REGION

REGION Network 243: DISABLE SAFETY AXIS NX15 13 ....18
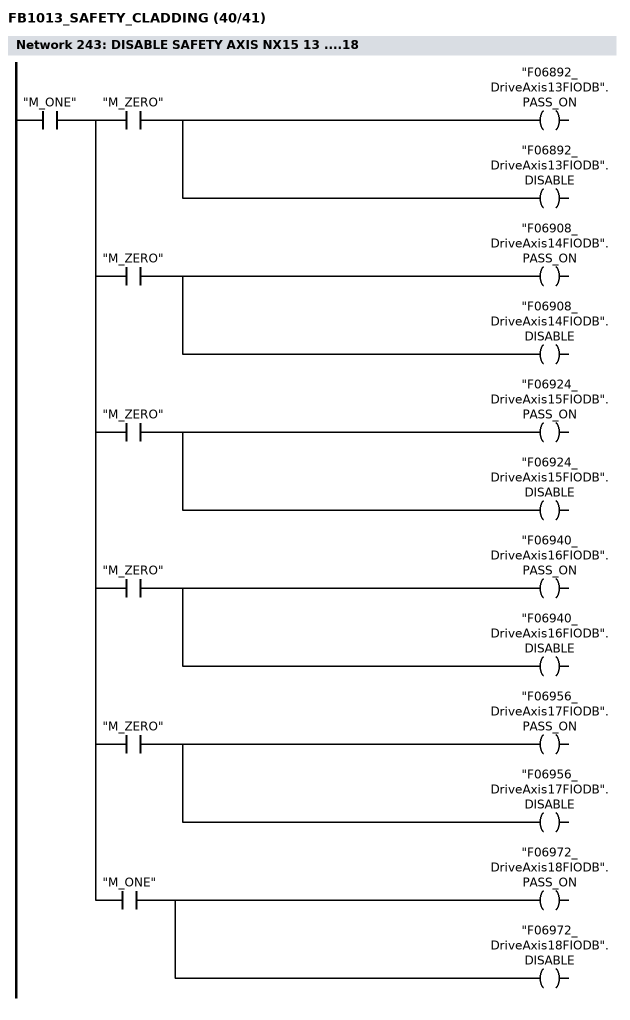
   RUNG wire#powerrail
      Contact( "M_ONE" )
      wire#w1
      Contact( "M_ZERO" )
      wire#w2
      Coil( "F06892_DriveAxis13FIODB".PASS_ON )
   END_RUNG
   RUNG wire#w2
      Coil( "F06892_DriveAxis13FIODB".DISABLE )
   END_RUNG
   RUNG wire#w1
      Contact( "M_ZERO" )
      wire#w3
      Coil( "F06908_DriveAxis14FIODB".PASS_ON )
   END_RUNG
   RUNG wire#w3
      Coil( "F06908_DriveAxis14FIODB".DISABLE )
   END_RUNG
   RUNG wire#w1
      Contact( "M_ZERO" )
      wire#w4
      Coil( "F06924_DriveAxis15FIODB".PASS_ON )
   END_RUNG
   RUNG wire#w4
      Coil( "F06924_DriveAxis15FIODB".DISABLE )
   END_RUNG
   RUNG wire#w1
      Contact( "M_ZERO" )
      wire#w5
      Coil( "F06940_DriveAxis16FIODB".PASS_ON )
   END_RUNG
   RUNG wire#w5
      Coil( "F06940_DriveAxis16FIODB".DISABLE )
   END_RUNG
   RUNG wire#w1
      Contact( "M_ZERO" )
      wire#w6
      Coil( "F06956_DriveAxis17FIODB".PASS_ON )
   END_RUNG
   RUNG wire#w6
      Coil( "F06956_DriveAxis17FIODB".DISABLE )
   END_RUNG
   RUNG wire#w1
      Contact( "M_ONE" )
      wire#w7
      Coil( "F06972_DriveAxis18FIODB".PASS_ON )
   END_RUNG
   RUNG wire#w7
      Coil( "F06972_DriveAxis18FIODB".DISABLE )
   END_RUNG
   // the same network as SCL:
   "F06892_DriveAxis13FIODB".PASS_ON := "M_ONE" AND "M_ZERO";
   "F06892_DriveAxis13FIODB".DISABLE := "F06892_DriveAxis13FIODB".PASS_ON;
   "F06908_DriveAxis14FIODB".PASS_ON := "M_ONE" AND "M_ZERO";
   "F06908_DriveAxis14FIODB".DISABLE := "F06908_DriveAxis14FIODB".PASS_ON;
   "F06924_DriveAxis15FIODB".PASS_ON := "M_ONE" AND "M_ZERO";
   "F06924_DriveAxis15FIODB".DISABLE := "F06924_DriveAxis15FIODB".PASS_ON;
   "F06940_DriveAxis16FIODB".PASS_ON := "M_ONE" AND "M_ZERO";
   "F06940_DriveAxis16FIODB".DISABLE := "F06940_DriveAxis16FIODB".PASS_ON;
   "F06956_DriveAxis17FIODB".PASS_ON := "M_ONE" AND "M_ZERO";
   "F06956_DriveAxis17FIODB".DISABLE := "F06956_DriveAxis17FIODB".PASS_ON;
   "F06972_DriveAxis18FIODB".PASS_ON := "M_ONE" AND "M_ONE";
   "F06972_DriveAxis18FIODB".DISABLE := "F06972_DriveAxis18FIODB".PASS_ON;
END_REGION

REGION Network 244: DISABLE SAFETY AXIS NX15 19 ....24
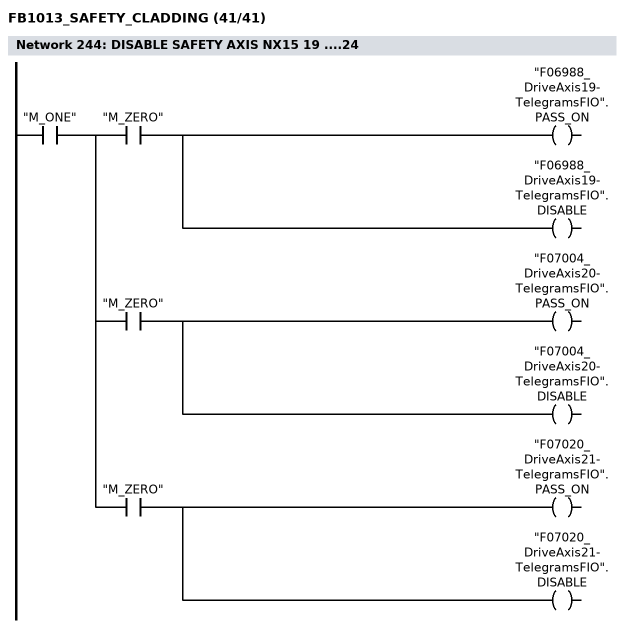
   RUNG wire#powerrail
      Contact( "M_ONE" )
      wire#w1
      Contact( "M_ZERO" )
      wire#w2
      Coil( "F06988_DriveAxis19-TelegramsFIO".PASS_ON )
   END_RUNG
   RUNG wire#w2
      Coil( "F06988_DriveAxis19-TelegramsFIO".DISABLE )
   END_RUNG
   RUNG wire#w1
      Contact( "M_ZERO" )
      wire#w3
      Coil( "F07004_DriveAxis20-TelegramsFIO".PASS_ON )
   END_RUNG
   RUNG wire#w3
      Coil( "F07004_DriveAxis20-TelegramsFIO".DISABLE )
   END_RUNG
   RUNG wire#w1
      Contact( "M_ZERO" )
      wire#w4
      Coil( "F07020_DriveAxis21-TelegramsFIO".PASS_ON )
   END_RUNG
   RUNG wire#w4
      Coil( "F07020_DriveAxis21-TelegramsFIO".DISABLE )
   END_RUNG
   // the same network as SCL:
   "F06988_DriveAxis19-TelegramsFIO".PASS_ON := "M_ONE" AND "M_ZERO";
   "F06988_DriveAxis19-TelegramsFIO".DISABLE := "F06988_DriveAxis19-TelegramsFIO".PASS_ON;
   "F07004_DriveAxis20-TelegramsFIO".PASS_ON := "M_ONE" AND "M_ZERO";
   "F07004_DriveAxis20-TelegramsFIO".DISABLE := "F07004_DriveAxis20-TelegramsFIO".PASS_ON;
   "F07020_DriveAxis21-TelegramsFIO".PASS_ON := "M_ONE" AND "M_ZERO";
   "F07020_DriveAxis21-TelegramsFIO".DISABLE := "F07020_DriveAxis21-TelegramsFIO".PASS_ON;
END_REGION
END_FUNCTION_BLOCK
